gfCNCPoint2[1220] = {X 302.9698, Y 48.2613, Z -2.1667, A 0.000, B 0.000, C 0.000 }
gfCNCPoint2[1221] = {X 302.3118, Y 47.6087, Z -2.1667, A 0.000, B 0.000, C 0.000 }
gfCNCPoint2[1222] = {X 301.8147, Y 46.8265, Z -2.1667, A 0.000, B 0.000, C 0.000 }
gfCNCPoint2[1223] = {X 301.5030, Y 45.9537, Z -2.1667, A 0.000, B 0.000, C 0.000 }
gfCNCPoint2[1224] = {X 301.3924, Y 45.0335, Z -2.1667, A 0.000, B 0.000, C 0.000 }
gfCNCPoint2[1225] = {X 301.3923, Y 44.2050, Z -2.1667, A 0.000, B 0.000, C 0.000 }
gfCNCPoint2[1226] = {X 301.5103, Y 43.2839, Z -2.1667, A 0.000, B 0.000, C 0.000 }
gfCNCPoint2[1227] = {X 301.8142, Y 42.4063, Z -2.1667, A 0.000, B 0.000, C 0.000 }
gfCNCPoint2[1228] = {X 302.2910, Y 41.6094, Z -2.1667, A 0.000, B 0.000, C 0.000 }
gfCNCPoint2[1229] = {X 302.9207, Y 40.9269, Z -2.1667, A 0.000, B 0.000, C 0.000 }
gfCNCPoint2[1230] = {X 302.9207, Y 33.8743, Z -2.1667, A 0.000, B 0.000, C 0.000 }
gfCNCPoint2[1231] = {X 293.6938, Y 33.8743, Z -2.1667, A 0.000, B 0.000, C 0.000 }
gfCNCPoint2[1232] = {X 293.6927, Y 40.9767, Z -2.1667, A 0.000, B 0.000, C 0.000 }
gfCNCPoint2[1233] = {X 294.3309, Y 41.6397, Z -2.1667, A 0.000, B 0.000, C 0.000 }
gfCNCPoint2[1234] = {X 294.8119, Y 42.4241, Z -2.1667, A 0.000, B 0.000, C 0.000 }
gfCNCPoint2[1235] = {X 295.1133, Y 43.2936, Z -2.1667, A 0.000, B 0.000, C 0.000 }
gfCNCPoint2[1236] = {X 295.2211, Y 44.2074, Z -2.1667, A 0.000, B 0.000, C 0.000 }
gfCNCPoint2[1237] = {X 295.2211, Y 45.0000, Z -2.1667, A 0.000, B 0.000, C 0.000 }
gfCNCPoint2[1238] = {X 295.1168, Y 45.9257, Z -2.1667, A 0.000, B 0.000, C 0.000 }
gfCNCPoint2[1239] = {X 294.8092, Y 46.8050, Z -2.1667, A 0.000, B 0.000, C 0.000 }
gfCNCPoint2[1240] = {X 294.3136, Y 47.5937, Z -2.1667, A 0.000, B 0.000, C 0.000 }
gfCNCPoint2[1241] = {X 293.6549, Y 48.2524, Z -2.1667, A 0.000, B 0.000, C 0.000 }
gfCNCPoint2[1242] = {X 292.8661, Y 48.7480, Z -2.1667, A 0.000, B 0.000, C 0.000 }
gfCNCPoint2[1243] = {X 291.9868, Y 49.0557, Z -2.1667, A 0.000, B 0.000, C 0.000 }
gfCNCPoint2[1244] = {X 291.0611, Y 49.1600, Z -2.1667, A 0.000, B 0.000, C 0.000 }
gfCNCPoint2[1245] = {X 284.6177, Y 49.1600, Z -2.1667, A 0.000, B 0.000, C 0.000 }
gfCNCPoint2[1246] = {X 283.6967, Y 49.0568, Z -2.1667, A 0.000, B 0.000, C 0.000 }
gfCNCPoint2[1247] = {X 282.8214, Y 48.7522, Z -2.1667, A 0.000, B 0.000, C 0.000 }
gfCNCPoint2[1248] = {X 282.0353, Y 48.2615, Z -2.1667, A 0.000, B 0.000, C 0.000 }
gfCNCPoint2[1249] = {X 281.3774, Y 47.6088, Z -2.1667, A 0.000, B 0.000, C 0.000 }
gfCNCPoint2[1250] = {X 280.8802, Y 46.8267, Z -2.1667, A 0.000, B 0.000, C 0.000 }
gfCNCPoint2[1251] = {X 280.5685, Y 45.9540, Z -2.1667, A 0.000, B 0.000, C 0.000 }
gfCNCPoint2[1252] = {X 280.4578, Y 45.0339, Z -2.1667, A 0.000, B 0.000, C 0.000 }
gfCNCPoint2[1253] = {X 280.4577, Y 44.2080, Z -2.1667, A 0.000, B 0.000, C 0.000 }
gfCNCPoint2[1254] = {X 280.5632, Y 43.2953, Z -2.1667, A 0.000, B 0.000, C 0.000 }
gfCNCPoint2[1255] = {X 280.8642, Y 42.4272, Z -2.1667, A 0.000, B 0.000, C 0.000 }
gfCNCPoint2[1256] = {X 281.3461, Y 41.6449, Z -2.1667, A 0.000, B 0.000, C 0.000 }
gfCNCPoint2[1257] = {X 281.9862, Y 40.9858, Z -2.1667, A 0.000, B 0.000, C 0.000 }
gfCNCPoint2[1258] = {X 281.9860, Y 28.5930, Z -2.1667, A 0.000, B 0.000, C 0.000 }
gfCNCPoint2[1259] = {X 277.9860, Y 28.5931, Z -2.1667, A 0.000, B 0.000, C 0.000 }
gfCNCPoint2[1260] = {X 282.0660, Y 28.5930, Z -2.1667, A 0.000, B 0.000, C 0.000 }
gfCNCPoint2[1261] = {X 282.0658, Y 16.1615, Z -2.1667, A 0.000, B 0.000, C 0.000 }
gfCNCPoint2[1262] = {X 281.4285, Y 15.5227, Z -2.1667, A 0.000, B 0.000, C 0.000 }
gfCNCPoint2[1263] = {X 280.9471, Y 14.7594, Z -2.1667, A 0.000, B 0.000, C 0.000 }
gfCNCPoint2[1264] = {X 280.6453, Y 13.9090, Z -2.1667, A 0.000, B 0.000, C 0.000 }
gfCNCPoint2[1265] = {X 280.5378, Y 13.0130, Z -2.1667, A 0.000, B 0.000, C 0.000 }
gfCNCPoint2[1266] = {X 280.5377, Y 12.1868, Z -2.1667, A 0.000, B 0.000, C 0.000 }
gfCNCPoint2[1267] = {X 280.6400, Y 11.2789, Z -2.1667, A 0.000, B 0.000, C 0.000 }
gfCNCPoint2[1268] = {X 280.9417, Y 10.4166, Z -2.1667, A 0.000, B 0.000, C 0.000 }
gfCNCPoint2[1269] = {X 281.4278, Y 9.6430, Z -2.1667, A 0.000, B 0.000, C 0.000 }
gfCNCPoint2[1270] = {X 282.0738, Y 8.9969, Z -2.1667, A 0.000, B 0.000, C 0.000 }
gfCNCPoint2[1271] = {X 282.8474, Y 8.5109, Z -2.1667, A 0.000, B 0.000, C 0.000 }
gfCNCPoint2[1272] = {X 283.7098, Y 8.2091, Z -2.1667, A 0.000, B 0.000, C 0.000 }
gfCNCPoint2[1273] = {X 284.6177, Y 8.1068, Z -2.1667, A 0.000, B 0.000, C 0.000 }
gfCNCPoint2[1274] = {X 291.0611, Y 8.1068, Z -2.1667, A 0.000, B 0.000, C 0.000 }
gfCNCPoint2[1275] = {X 291.9690, Y 8.2091, Z -2.1667, A 0.000, B 0.000, C 0.000 }
gfCNCPoint2[1276] = {X 292.8314, Y 8.5109, Z -2.1667, A 0.000, B 0.000, C 0.000 }
gfCNCPoint2[1277] = {X 293.6050, Y 8.9969, Z -2.1667, A 0.000, B 0.000, C 0.000 }
gfCNCPoint2[1278] = {X 294.2510, Y 9.6430, Z -2.1667, A 0.000, B 0.000, C 0.000 }
gfCNCPoint2[1279] = {X 294.7371, Y 10.4166, Z -2.1667, A 0.000, B 0.000, C 0.000 }
gfCNCPoint2[1280] = {X 295.0388, Y 11.2789, Z -2.1667, A 0.000, B 0.000, C 0.000 }
gfCNCPoint2[1281] = {X 295.1411, Y 12.1868, Z -2.1667, A 0.000, B 0.000, C 0.000 }
gfCNCPoint2[1282] = {X 295.1411, Y 12.9781, Z -2.1667, A 0.000, B 0.000, C 0.000 }
gfCNCPoint2[1283] = {X 295.0472, Y 13.8483, Z -2.1667, A 0.000, B 0.000, C 0.000 }
gfCNCPoint2[1284] = {X 294.7699, Y 14.6784, Z -2.1667, A 0.000, B 0.000, C 0.000 }
gfCNCPoint2[1285] = {X 294.3219, Y 15.4303, Z -2.1667, A 0.000, B 0.000, C 0.000 }
gfCNCPoint2[1286] = {X 293.7238, Y 16.0694, Z -2.1667, A 0.000, B 0.000, C 0.000 }
gfCNCPoint2[1287] = {X 293.6665, Y 16.1178, Z -2.1667, A 0.000, B 0.000, C 0.000 }
gfCNCPoint2[1288] = {X 293.6084, Y 16.1652, Z -2.1667, A 0.000, B 0.000, C 0.000 }
gfCNCPoint2[1289] = {X 293.6127, Y 16.1999, Z -2.1667, A 0.000, B 0.000, C 0.000 }
gfCNCPoint2[1290] = {X 293.6140, Y 22.4371, Z -2.1667, A 0.000, B 0.000, C 0.000 }
gfCNCPoint2[1291] = {X 293.7675, Y 22.4365, Z -2.1667, A 0.000, B 0.000, C 0.000 }
gfCNCPoint2[1292] = {X 302.9997, Y 22.4365, Z -2.1667, A 0.000, B 0.000, C 0.000 }
gfCNCPoint2[1293] = {X 303.0047, Y 16.1649, Z -2.1667, A 0.000, B 0.000, C 0.000 }
gfCNCPoint2[1294] = {X 302.9465, Y 16.1175, Z -2.1667, A 0.000, B 0.000, C 0.000 }
gfCNCPoint2[1295] = {X 302.8892, Y 16.0690, Z -2.1667, A 0.000, B 0.000, C 0.000 }
gfCNCPoint2[1296] = {X 302.2967, Y 15.4373, Z -2.1667, A 0.000, B 0.000, C 0.000 }
gfCNCPoint2[1297] = {X 301.8510, Y 14.6947, Z -2.1667, A 0.000, B 0.000, C 0.000 }
gfCNCPoint2[1298] = {X 301.5720, Y 13.8747, Z -2.1667, A 0.000, B 0.000, C 0.000 }
gfCNCPoint2[1299] = {X 301.4724, Y 13.0144, Z -2.1667, A 0.000, B 0.000, C 0.000 }
gfCNCPoint2[1300] = {X 301.4723, Y 12.1868, Z -2.1667, A 0.000, B 0.000, C 0.000 }
gfCNCPoint2[1301] = {X 301.5745, Y 11.2789, Z -2.1667, A 0.000, B 0.000, C 0.000 }
gfCNCPoint2[1302] = {X 301.8763, Y 10.4166, Z -2.1667, A 0.000, B 0.000, C 0.000 }
gfCNCPoint2[1303] = {X 302.3624, Y 9.6430, Z -2.1667, A 0.000, B 0.000, C 0.000 }
gfCNCPoint2[1304] = {X 303.0084, Y 8.9969, Z -2.1667, A 0.000, B 0.000, C 0.000 }
gfCNCPoint2[1305] = {X 303.7820, Y 8.5109, Z -2.1667, A 0.000, B 0.000, C 0.000 }
gfCNCPoint2[1306] = {X 304.6444, Y 8.2091, Z -2.1667, A 0.000, B 0.000, C 0.000 }
gfCNCPoint2[1307] = {X 305.5523, Y 8.1068, Z -2.1667, A 0.000, B 0.000, C 0.000 }
gfCNCPoint2[1308] = {X 311.9957, Y 8.1068, Z -2.1667, A 0.000, B 0.000, C 0.000 }
gfCNCPoint2[1309] = {X 312.9036, Y 8.2091, Z -2.1667, A 0.000, B 0.000, C 0.000 }
gfCNCPoint2[1310] = {X 313.7660, Y 8.5109, Z -2.1667, A 0.000, B 0.000, C 0.000 }
gfCNCPoint2[1311] = {X 314.5396, Y 8.9969, Z -2.1667, A 0.000, B 0.000, C 0.000 }
gfCNCPoint2[1312] = {X 315.1856, Y 9.6430, Z -2.1667, A 0.000, B 0.000, C 0.000 }
gfCNCPoint2[1313] = {X 315.6717, Y 10.4166, Z -2.1667, A 0.000, B 0.000, C 0.000 }
gfCNCPoint2[1314] = {X 315.9734, Y 11.2789, Z -2.1667, A 0.000, B 0.000, C 0.000 }
gfCNCPoint2[1315] = {X 316.0757, Y 12.1868, Z -2.1667, A 0.000, B 0.000, C 0.000 }
gfCNCPoint2[1316] = {X 316.0757, Y 12.9781, Z -2.1667, A 0.000, B 0.000, C 0.000 }
gfCNCPoint2[1317] = {X 315.9818, Y 13.8483, Z -2.1667, A 0.000, B 0.000, C 0.000 }
gfCNCPoint2[1318] = {X 315.7045, Y 14.6784, Z -2.1667, A 0.000, B 0.000, C 0.000 }
gfCNCPoint2[1319] = {X 315.2566, Y 15.4302, Z -2.1667, A 0.000, B 0.000, C 0.000 }
gfCNCPoint2[1320] = {X 314.6586, Y 16.0692, Z -2.1667, A 0.000, B 0.000, C 0.000 }
gfCNCPoint2[1321] = {X 314.6041, Y 16.1153, Z -2.1667, A 0.000, B 0.000, C 0.000 }
gfCNCPoint2[1322] = {X 314.5488, Y 16.1605, Z -2.1667, A 0.000, B 0.000, C 0.000 }
gfCNCPoint2[1323] = {X 314.5472, Y 41.0281, Z -2.1667, A 0.000, B 0.000, C 0.000 }
gfCNCPoint2[1324] = {X 314.6336, Y 41.0962, Z -2.1667, A 0.000, B 0.000, C 0.000 }
gfCNCPoint2[1325] = {X 315.2363, Y 41.7299, Z -2.1667, A 0.000, B 0.000, C 0.000 }
gfCNCPoint2[1326] = {X 315.6902, Y 42.4775, Z -2.1667, A 0.000, B 0.000, C 0.000 }
gfCNCPoint2[1327] = {X 315.9743, Y 43.3047, Z -2.1667, A 0.000, B 0.000, C 0.000 }
gfCNCPoint2[1328] = {X 316.0756, Y 44.1734, Z -2.1667, A 0.000, B 0.000, C 0.000 }
gfCNCPoint2[1329] = {X 316.0757, Y 45.0000, Z -2.1667, A 0.000, B 0.000, C 0.000 }
gfCNCPoint2[1330] = {X 315.9734, Y 45.9079, Z -2.1667, A 0.000, B 0.000, C 0.000 }
gfCNCPoint2[1331] = {X 315.6717, Y 46.7702, Z -2.1667, A 0.000, B 0.000, C 0.000 }
gfCNCPoint2[1332] = {X 315.1856, Y 47.5438, Z -2.1667, A 0.000, B 0.000, C 0.000 }
gfCNCPoint2[1333] = {X 314.5396, Y 48.1899, Z -2.1667, A 0.000, B 0.000, C 0.000 }
gfCNCPoint2[1334] = {X 313.7660, Y 48.6760, Z -2.1667, A 0.000, B 0.000, C 0.000 }
gfCNCPoint2[1335] = {X 312.9036, Y 48.9777, Z -2.1667, A 0.000, B 0.000, C 0.000 }
gfCNCPoint2[1336] = {X 311.9957, Y 49.0800, Z -2.1667, A 0.000, B 0.000, C 0.000 }
gfCNCPoint2[1337] = {X 305.5523, Y 49.0800, Z -2.1667, A 0.000, B 0.000, C 0.000 }
gfCNCPoint2[1338] = {X 304.6489, Y 48.9787, Z -2.1667, A 0.000, B 0.000, C 0.000 }
gfCNCPoint2[1339] = {X 303.7905, Y 48.6800, Z -2.1667, A 0.000, B 0.000, C 0.000 }
gfCNCPoint2[1340] = {X 303.0194, Y 48.1986, Z -2.1667, A 0.000, B 0.000, C 0.000 }
gfCNCPoint2[1341] = {X 302.3741, Y 47.5585, Z -2.1667, A 0.000, B 0.000, C 0.000 }
gfCNCPoint2[1342] = {X 301.8865, Y 46.7914, Z -2.1667, A 0.000, B 0.000, C 0.000 }
gfCNCPoint2[1343] = {X 301.5809, Y 45.9353, Z -2.1667, A 0.000, B 0.000, C 0.000 }
gfCNCPoint2[1344] = {X 301.4724, Y 45.0328, Z -2.1667, A 0.000, B 0.000, C 0.000 }
gfCNCPoint2[1345] = {X 301.4723, Y 44.2070, Z -2.1667, A 0.000, B 0.000, C 0.000 }
gfCNCPoint2[1346] = {X 301.5903, Y 43.2934, Z -2.1667, A 0.000, B 0.000, C 0.000 }
gfCNCPoint2[1347] = {X 301.8943, Y 42.4238, Z -2.1667, A 0.000, B 0.000, C 0.000 }
gfCNCPoint2[1348] = {X 302.3713, Y 41.6358, Z -2.1667, A 0.000, B 0.000, C 0.000 }
gfCNCPoint2[1349] = {X 303.0007, Y 40.9632, Z -2.1667, A 0.000, B 0.000, C 0.000 }
gfCNCPoint2[1350] = {X 303.0007, Y 33.7943, Z -2.1667, A 0.000, B 0.000, C 0.000 }
gfCNCPoint2[1351] = {X 293.6138, Y 33.7943, Z -2.1667, A 0.000, B 0.000, C 0.000 }
gfCNCPoint2[1352] = {X 293.6127, Y 41.0143, Z -2.1667, A 0.000, B 0.000, C 0.000 }
gfCNCPoint2[1353] = {X 294.2505, Y 41.6665, Z -2.1667, A 0.000, B 0.000, C 0.000 }
gfCNCPoint2[1354] = {X 294.7316, Y 42.4415, Z -2.1667, A 0.000, B 0.000, C 0.000 }
gfCNCPoint2[1355] = {X 295.0333, Y 43.3024, Z -2.1667, A 0.000, B 0.000, C 0.000 }
gfCNCPoint2[1356] = {X 295.1411, Y 44.2082, Z -2.1667, A 0.000, B 0.000, C 0.000 }
gfCNCPoint2[1357] = {X 295.1411, Y 45.0000, Z -2.1667, A 0.000, B 0.000, C 0.000 }
gfCNCPoint2[1358] = {X 295.0388, Y 45.9079, Z -2.1667, A 0.000, B 0.000, C 0.000 }
gfCNCPoint2[1359] = {X 294.7371, Y 46.7702, Z -2.1667, A 0.000, B 0.000, C 0.000 }
gfCNCPoint2[1360] = {X 294.2510, Y 47.5438, Z -2.1667, A 0.000, B 0.000, C 0.000 }
gfCNCPoint2[1361] = {X 293.6050, Y 48.1899, Z -2.1667, A 0.000, B 0.000, C 0.000 }
gfCNCPoint2[1362] = {X 292.8314, Y 48.6760, Z -2.1667, A 0.000, B 0.000, C 0.000 }
gfCNCPoint2[1363] = {X 291.9690, Y 48.9777, Z -2.1667, A 0.000, B 0.000, C 0.000 }
gfCNCPoint2[1364] = {X 291.0611, Y 49.0800, Z -2.1667, A 0.000, B 0.000, C 0.000 }
gfCNCPoint2[1365] = {X 284.6177, Y 49.0800, Z -2.1667, A 0.000, B 0.000, C 0.000 }
gfCNCPoint2[1366] = {X 283.7144, Y 48.9788, Z -2.1667, A 0.000, B 0.000, C 0.000 }
gfCNCPoint2[1367] = {X 282.8560, Y 48.6801, Z -2.1667, A 0.000, B 0.000, C 0.000 }
gfCNCPoint2[1368] = {X 282.0850, Y 48.1987, Z -2.1667, A 0.000, B 0.000, C 0.000 }
gfCNCPoint2[1369] = {X 281.4397, Y 47.5587, Z -2.1667, A 0.000, B 0.000, C 0.000 }
gfCNCPoint2[1370] = {X 280.9521, Y 46.7916, Z -2.1667, A 0.000, B 0.000, C 0.000 }
gfCNCPoint2[1371] = {X 280.6464, Y 45.9356, Z -2.1667, A 0.000, B 0.000, C 0.000 }
gfCNCPoint2[1372] = {X 280.5378, Y 45.0332, Z -2.1667, A 0.000, B 0.000, C 0.000 }
gfCNCPoint2[1373] = {X 280.5377, Y 44.2084, Z -2.1667, A 0.000, B 0.000, C 0.000 }
gfCNCPoint2[1374] = {X 280.6433, Y 43.3039, Z -2.1667, A 0.000, B 0.000, C 0.000 }
gfCNCPoint2[1375] = {X 280.9445, Y 42.4445, Z -2.1667, A 0.000, B 0.000, C 0.000 }
gfCNCPoint2[1376] = {X 281.4266, Y 41.6719, Z -2.1667, A 0.000, B 0.000, C 0.000 }
gfCNCPoint2[1377] = {X 282.0662, Y 41.0237, Z -2.1667, A 0.000, B 0.000, C 0.000 }
gfCNCPoint2[1378] = {X 282.0660, Y 28.5930, Z -2.1667, A 0.000, B 0.000, C 0.000 }
gfCNCPoint2[1379] = {X 278.0660, Y 28.5931, Z -2.1667, A 0.000, B 0.000, C 0.000 }
gfCNCPoint2[1380] = {X 282.1460, Y 28.5930, Z -2.1667, A 0.000, B 0.000, C 0.000 }
gfCNCPoint2[1381] = {X 282.1458, Y 16.1228, Z -2.1667, A 0.000, B 0.000, C 0.000 }
gfCNCPoint2[1382] = {X 281.5036, Y 15.4885, Z -2.1667, A 0.000, B 0.000, C 0.000 }
gfCNCPoint2[1383] = {X 281.0199, Y 14.7262, Z -2.1667, A 0.000, B 0.000, C 0.000 }
gfCNCPoint2[1384] = {X 280.7195, Y 13.8749, Z -2.1667, A 0.000, B 0.000, C 0.000 }
gfCNCPoint2[1385] = {X 280.6177, Y 12.9779, Z -2.1667, A 0.000, B 0.000, C 0.000 }
gfCNCPoint2[1386] = {X 280.6177, Y 12.1868, Z -2.1667, A 0.000, B 0.000, C 0.000 }
gfCNCPoint2[1387] = {X 280.7180, Y 11.2967, Z -2.1667, A 0.000, B 0.000, C 0.000 }
gfCNCPoint2[1388] = {X 281.0138, Y 10.4513, Z -2.1667, A 0.000, B 0.000, C 0.000 }
gfCNCPoint2[1389] = {X 281.4903, Y 9.6929, Z -2.1667, A 0.000, B 0.000, C 0.000 }
gfCNCPoint2[1390] = {X 282.1237, Y 9.0595, Z -2.1667, A 0.000, B 0.000, C 0.000 }
gfCNCPoint2[1391] = {X 282.8821, Y 8.5829, Z -2.1667, A 0.000, B 0.000, C 0.000 }
gfCNCPoint2[1392] = {X 283.7276, Y 8.2871, Z -2.1667, A 0.000, B 0.000, C 0.000 }
gfCNCPoint2[1393] = {X 284.6177, Y 8.1868, Z -2.1667, A 0.000, B 0.000, C 0.000 }
gfCNCPoint2[1394] = {X 291.0611, Y 8.1868, Z -2.1667, A 0.000, B 0.000, C 0.000 }
gfCNCPoint2[1395] = {X 291.9512, Y 8.2871, Z -2.1667, A 0.000, B 0.000, C 0.000 }
gfCNCPoint2[1396] = {X 292.7967, Y 8.5829, Z -2.1667, A 0.000, B 0.000, C 0.000 }
gfCNCPoint2[1397] = {X 293.5551, Y 9.0595, Z -2.1667, A 0.000, B 0.000, C 0.000 }
gfCNCPoint2[1398] = {X 294.1885, Y 9.6929, Z -2.1667, A 0.000, B 0.000, C 0.000 }
gfCNCPoint2[1399] = {X 294.6650, Y 10.4513, Z -2.1667, A 0.000, B 0.000, C 0.000 }
gfCNCPoint2[1400] = {X 294.9608, Y 11.2967, Z -2.1667, A 0.000, B 0.000, C 0.000 }
gfCNCPoint2[1401] = {X 295.0611, Y 12.1868, Z -2.1667, A 0.000, B 0.000, C 0.000 }
gfCNCPoint2[1402] = {X 295.0609, Y 13.0192, Z -2.1667, A 0.000, B 0.000, C 0.000 }
gfCNCPoint2[1403] = {X 294.9624, Y 13.8613, Z -2.1667, A 0.000, B 0.000, C 0.000 }
gfCNCPoint2[1404] = {X 294.6886, Y 14.6637, Z -2.1667, A 0.000, B 0.000, C 0.000 }
gfCNCPoint2[1405] = {X 294.2518, Y 15.3904, Z -2.1667, A 0.000, B 0.000, C 0.000 }
gfCNCPoint2[1406] = {X 293.6716, Y 16.0087, Z -2.1667, A 0.000, B 0.000, C 0.000 }
gfCNCPoint2[1407] = {X 293.5954, Y 16.0727, Z -2.1667, A 0.000, B 0.000, C 0.000 }
gfCNCPoint2[1408] = {X 293.5177, Y 16.1348, Z -2.1667, A 0.000, B 0.000, C 0.000 }
gfCNCPoint2[1409] = {X 293.5327, Y 16.1919, Z -2.1667, A 0.000, B 0.000, C 0.000 }
gfCNCPoint2[1410] = {X 293.5341, Y 22.5174, Z -2.1667, A 0.000, B 0.000, C 0.000 }
gfCNCPoint2[1411] = {X 293.7676, Y 22.5165, Z -2.1667, A 0.000, B 0.000, C 0.000 }
gfCNCPoint2[1412] = {X 303.0796, Y 22.5177, Z -2.1667, A 0.000, B 0.000, C 0.000 }
gfCNCPoint2[1413] = {X 303.0803, Y 16.1920, Z -2.1667, A 0.000, B 0.000, C 0.000 }
gfCNCPoint2[1414] = {X 303.0955, Y 16.1346, Z -2.1667, A 0.000, B 0.000, C 0.000 }
gfCNCPoint2[1415] = {X 303.0176, Y 16.0725, Z -2.1667, A 0.000, B 0.000, C 0.000 }
gfCNCPoint2[1416] = {X 302.9414, Y 16.0084, Z -2.1667, A 0.000, B 0.000, C 0.000 }
gfCNCPoint2[1417] = {X 302.3552, Y 15.3819, Z -2.1667, A 0.000, B 0.000, C 0.000 }
gfCNCPoint2[1418] = {X 301.9161, Y 14.6448, Z -2.1667, A 0.000, B 0.000, C 0.000 }
gfCNCPoint2[1419] = {X 301.6443, Y 13.8310, Z -2.1667, A 0.000, B 0.000, C 0.000 }
gfCNCPoint2[1420] = {X 301.5523, Y 12.9779, Z -2.1667, A 0.000, B 0.000, C 0.000 }
gfCNCPoint2[1421] = {X 301.5523, Y 12.1868, Z -2.1667, A 0.000, B 0.000, C 0.000 }
gfCNCPoint2[1422] = {X 301.6525, Y 11.2967, Z -2.1667, A 0.000, B 0.000, C 0.000 }
gfCNCPoint2[1423] = {X 301.9484, Y 10.4513, Z -2.1667, A 0.000, B 0.000, C 0.000 }
gfCNCPoint2[1424] = {X 302.4249, Y 9.6929, Z -2.1667, A 0.000, B 0.000, C 0.000 }
gfCNCPoint2[1425] = {X 303.0583, Y 9.0595, Z -2.1667, A 0.000, B 0.000, C 0.000 }
gfCNCPoint2[1426] = {X 303.8167, Y 8.5829, Z -2.1667, A 0.000, B 0.000, C 0.000 }
gfCNCPoint2[1427] = {X 304.6622, Y 8.2871, Z -2.1667, A 0.000, B 0.000, C 0.000 }
gfCNCPoint2[1428] = {X 305.5523, Y 8.1868, Z -2.1667, A 0.000, B 0.000, C 0.000 }
gfCNCPoint2[1429] = {X 311.9957, Y 8.1868, Z -2.1667, A 0.000, B 0.000, C 0.000 }
gfCNCPoint2[1430] = {X 312.8858, Y 8.2871, Z -2.1667, A 0.000, B 0.000, C 0.000 }
gfCNCPoint2[1431] = {X 313.7313, Y 8.5829, Z -2.1667, A 0.000, B 0.000, C 0.000 }
gfCNCPoint2[1432] = {X 314.4897, Y 9.0595, Z -2.1667, A 0.000, B 0.000, C 0.000 }
gfCNCPoint2[1433] = {X 315.1230, Y 9.6929, Z -2.1667, A 0.000, B 0.000, C 0.000 }
gfCNCPoint2[1434] = {X 315.5996, Y 10.4513, Z -2.1667, A 0.000, B 0.000, C 0.000 }
gfCNCPoint2[1435] = {X 315.8954, Y 11.2967, Z -2.1667, A 0.000, B 0.000, C 0.000 }
gfCNCPoint2[1436] = {X 315.9957, Y 12.1868, Z -2.1667, A 0.000, B 0.000, C 0.000 }
gfCNCPoint2[1437] = {X 315.9955, Y 13.0192, Z -2.1667, A 0.000, B 0.000, C 0.000 }
gfCNCPoint2[1438] = {X 315.8970, Y 13.8613, Z -2.1667, A 0.000, B 0.000, C 0.000 }
gfCNCPoint2[1439] = {X 315.6232, Y 14.6637, Z -2.1667, A 0.000, B 0.000, C 0.000 }
gfCNCPoint2[1440] = {X 315.1865, Y 15.3903, Z -2.1667, A 0.000, B 0.000, C 0.000 }
gfCNCPoint2[1441] = {X 314.6064, Y 16.0086, Z -2.1667, A 0.000, B 0.000, C 0.000 }
gfCNCPoint2[1442] = {X 314.5386, Y 16.0657, Z -2.1667, A 0.000, B 0.000, C 0.000 }
gfCNCPoint2[1443] = {X 314.4695, Y 16.1213, Z -2.1667, A 0.000, B 0.000, C 0.000 }
gfCNCPoint2[1444] = {X 314.4674, Y 16.3117, Z -2.1667, A 0.000, B 0.000, C 0.000 }
gfCNCPoint2[1445] = {X 314.4672, Y 41.0669, Z -2.1667, A 0.000, B 0.000, C 0.000 }
gfCNCPoint2[1446] = {X 314.6061, Y 41.1780, Z -2.1667, A 0.000, B 0.000, C 0.000 }
gfCNCPoint2[1447] = {X 315.1925, Y 41.8046, Z -2.1667, A 0.000, B 0.000, C 0.000 }
gfCNCPoint2[1448] = {X 315.6318, Y 42.5418, Z -2.1667, A 0.000, B 0.000, C 0.000 }
gfCNCPoint2[1449] = {X 315.9037, Y 43.3557, Z -2.1667, A 0.000, B 0.000, C 0.000 }
gfCNCPoint2[1450] = {X 315.9957, Y 44.2089, Z -2.1667, A 0.000, B 0.000, C 0.000 }
gfCNCPoint2[1451] = {X 315.9957, Y 45.0000, Z -2.1667, A 0.000, B 0.000, C 0.000 }
gfCNCPoint2[1452] = {X 315.8954, Y 45.8901, Z -2.1667, A 0.000, B 0.000, C 0.000 }
gfCNCPoint2[1453] = {X 315.5996, Y 46.7355, Z -2.1667, A 0.000, B 0.000, C 0.000 }
gfCNCPoint2[1454] = {X 315.1230, Y 47.4940, Z -2.1667, A 0.000, B 0.000, C 0.000 }
gfCNCPoint2[1455] = {X 314.4897, Y 48.1273, Z -2.1667, A 0.000, B 0.000, C 0.000 }
gfCNCPoint2[1456] = {X 313.7313, Y 48.6039, Z -2.1667, A 0.000, B 0.000, C 0.000 }
gfCNCPoint2[1457] = {X 312.8858, Y 48.8997, Z -2.1667, A 0.000, B 0.000, C 0.000 }
gfCNCPoint2[1458] = {X 311.9957, Y 49.0000, Z -2.1667, A 0.000, B 0.000, C 0.000 }
gfCNCPoint2[1459] = {X 305.5523, Y 49.0000, Z -2.1667, A 0.000, B 0.000, C 0.000 }
gfCNCPoint2[1460] = {X 304.6622, Y 48.8997, Z -2.1667, A 0.000, B 0.000, C 0.000 }
gfCNCPoint2[1461] = {X 303.8167, Y 48.6039, Z -2.1667, A 0.000, B 0.000, C 0.000 }
gfCNCPoint2[1462] = {X 303.0583, Y 48.1273, Z -2.1667, A 0.000, B 0.000, C 0.000 }
gfCNCPoint2[1463] = {X 302.4249, Y 47.4939, Z -2.1667, A 0.000, B 0.000, C 0.000 }
gfCNCPoint2[1464] = {X 301.9484, Y 46.7355, Z -2.1667, A 0.000, B 0.000, C 0.000 }
gfCNCPoint2[1465] = {X 301.6525, Y 45.8900, Z -2.1667, A 0.000, B 0.000, C 0.000 }
gfCNCPoint2[1466] = {X 301.5523, Y 45.0000, Z -2.1667, A 0.000, B 0.000, C 0.000 }
gfCNCPoint2[1467] = {X 301.5523, Y 44.2089, Z -2.1667, A 0.000, B 0.000, C 0.000 }
gfCNCPoint2[1468] = {X 301.6702, Y 43.3029, Z -2.1667, A 0.000, B 0.000, C 0.000 }
gfCNCPoint2[1469] = {X 301.9745, Y 42.4415, Z -2.1667, A 0.000, B 0.000, C 0.000 }
gfCNCPoint2[1470] = {X 302.4516, Y 41.6624, Z -2.1667, A 0.000, B 0.000, C 0.000 }
gfCNCPoint2[1471] = {X 303.0807, Y 40.9999, Z -2.1667, A 0.000, B 0.000, C 0.000 }
gfCNCPoint2[1472] = {X 303.0807, Y 33.7143, Z -2.1667, A 0.000, B 0.000, C 0.000 }
gfCNCPoint2[1473] = {X 293.9337, Y 33.7143, Z -2.1667, A 0.000, B 0.000, C 0.000 }
gfCNCPoint2[1474] = {X 293.5338, Y 33.7132, Z -2.1667, A 0.000, B 0.000, C 0.000 }
gfCNCPoint2[1475] = {X 293.5327, Y 41.0524, Z -2.1667, A 0.000, B 0.000, C 0.000 }
gfCNCPoint2[1476] = {X 294.1700, Y 41.6937, Z -2.1667, A 0.000, B 0.000, C 0.000 }
gfCNCPoint2[1477] = {X 294.6513, Y 42.4591, Z -2.1667, A 0.000, B 0.000, C 0.000 }
gfCNCPoint2[1478] = {X 294.9532, Y 43.3113, Z -2.1667, A 0.000, B 0.000, C 0.000 }
gfCNCPoint2[1479] = {X 295.0611, Y 44.2089, Z -2.1667, A 0.000, B 0.000, C 0.000 }
gfCNCPoint2[1480] = {X 295.0611, Y 45.0000, Z -2.1667, A 0.000, B 0.000, C 0.000 }
gfCNCPoint2[1481] = {X 294.9608, Y 45.8901, Z -2.1667, A 0.000, B 0.000, C 0.000 }
gfCNCPoint2[1482] = {X 294.6650, Y 46.7355, Z -2.1667, A 0.000, B 0.000, C 0.000 }
gfCNCPoint2[1483] = {X 294.1885, Y 47.4940, Z -2.1667, A 0.000, B 0.000, C 0.000 }
gfCNCPoint2[1484] = {X 293.5551, Y 48.1273, Z -2.1667, A 0.000, B 0.000, C 0.000 }
gfCNCPoint2[1485] = {X 292.7967, Y 48.6039, Z -2.1667, A 0.000, B 0.000, C 0.000 }
gfCNCPoint2[1486] = {X 291.9512, Y 48.8997, Z -2.1667, A 0.000, B 0.000, C 0.000 }
gfCNCPoint2[1487] = {X 291.0611, Y 49.0000, Z -2.1667, A 0.000, B 0.000, C 0.000 }
gfCNCPoint2[1488] = {X 284.6177, Y 49.0000, Z -2.1667, A 0.000, B 0.000, C 0.000 }
gfCNCPoint2[1489] = {X 283.7276, Y 48.8997, Z -2.1667, A 0.000, B 0.000, C 0.000 }
gfCNCPoint2[1490] = {X 282.8821, Y 48.6039, Z -2.1667, A 0.000, B 0.000, C 0.000 }
gfCNCPoint2[1491] = {X 282.1237, Y 48.1273, Z -2.1667, A 0.000, B 0.000, C 0.000 }
gfCNCPoint2[1492] = {X 281.4903, Y 47.4939, Z -2.1667, A 0.000, B 0.000, C 0.000 }
gfCNCPoint2[1493] = {X 281.0138, Y 46.7355, Z -2.1667, A 0.000, B 0.000, C 0.000 }
gfCNCPoint2[1494] = {X 280.7179, Y 45.8900, Z -2.1667, A 0.000, B 0.000, C 0.000 }
gfCNCPoint2[1495] = {X 280.6177, Y 45.0000, Z -2.1667, A 0.000, B 0.000, C 0.000 }
gfCNCPoint2[1496] = {X 280.6177, Y 44.2089, Z -2.1667, A 0.000, B 0.000, C 0.000 }
gfCNCPoint2[1497] = {X 280.7234, Y 43.3127, Z -2.1667, A 0.000, B 0.000, C 0.000 }
gfCNCPoint2[1498] = {X 281.0249, Y 42.4620, Z -2.1667, A 0.000, B 0.000, C 0.000 }
gfCNCPoint2[1499] = {X 281.5071, Y 41.6992, Z -2.1667, A 0.000, B 0.000, C 0.000 }
gfCNCPoint2[1500] = {X 282.1462, Y 41.0620, Z -2.1667, A 0.000, B 0.000, C 0.000 }
gfCNCPoint2[1501] = {X 282.1460, Y 28.5930, Z -2.1667, A 0.000, B 0.000, C 0.000 }
gfCNCPoint2[1502] = {X 278.0660, Y 28.5931, Z -2.1667, A 0.000, B 0.000, C 0.000 }
gfCNCPoint2[1503] = {X 278.0660, Y 28.5931, Z 0.8333, A 0.000, B 0.000, C 0.000 }
gfCNCPoint2[1504] = {X 278.0660, Y 28.5931, Z 11.0000, A 0.000, B 0.000, C 0.000 }
gfCNCPoint2[1505] = {X 353.3541, Y 107.0427, Z 11.0000, A 0.000, B 0.000, C 0.000 }
gfCNCPoint2[1506] = {X 353.3541, Y 107.0427, Z 0.8333, A 0.000, B 0.000, C 0.000 }
gfCNCPoint2[1507] = {X 353.3541, Y 107.0427, Z -2.1667, A 0.000, B 0.000, C 0.000 }
gfCNCPoint2[1508] = {X 353.2424, Y 102.9642, Z -2.1667, A 0.000, B 0.000, C 0.000 }
gfCNCPoint2[1509] = {X 347.7202, Y 103.0327, Z -2.1667, A 0.000, B 0.000, C 0.000 }
gfCNCPoint2[1510] = {X 342.1984, Y 102.9360, Z -2.1667, A 0.000, B 0.000, C 0.000 }
gfCNCPoint2[1511] = {X 336.6820, Y 102.6741, Z -2.1667, A 0.000, B 0.000, C 0.000 }
gfCNCPoint2[1512] = {X 333.1921, Y 102.3991, Z -2.1667, A 0.000, B 0.000, C 0.000 }
gfCNCPoint2[1513] = {X 329.7159, Y 101.9862, Z -2.1667, A 0.000, B 0.000, C 0.000 }
gfCNCPoint2[1514] = {X 326.2587, Y 101.4359, Z -2.1667, A 0.000, B 0.000, C 0.000 }
gfCNCPoint2[1515] = {X 323.4092, Y 100.8312, Z -2.1667, A 0.000, B 0.000, C 0.000 }
gfCNCPoint2[1516] = {X 320.6119, Y 100.0183, Z -2.1667, A 0.000, B 0.000, C 0.000 }
gfCNCPoint2[1517] = {X 317.8822, Y 99.0016, Z -2.1667, A 0.000, B 0.000, C 0.000 }
gfCNCPoint2[1518] = {X 316.3696, Y 98.3034, Z -2.1667, A 0.000, B 0.000, C 0.000 }
gfCNCPoint2[1519] = {X 314.9205, Y 97.4815, Z -2.1667, A 0.000, B 0.000, C 0.000 }
gfCNCPoint2[1520] = {X 313.5450, Y 96.5415, Z -2.1667, A 0.000, B 0.000, C 0.000 }
gfCNCPoint2[1521] = {X 312.2527, Y 95.4901, Z -2.1667, A 0.000, B 0.000, C 0.000 }
gfCNCPoint2[1522] = {X 311.2490, Y 94.4920, Z -2.1667, A 0.000, B 0.000, C 0.000 }
gfCNCPoint2[1523] = {X 310.3708, Y 93.3817, Z -2.1667, A 0.000, B 0.000, C 0.000 }
gfCNCPoint2[1524] = {X 309.6305, Y 92.1752, Z -2.1667, A 0.000, B 0.000, C 0.000 }
gfCNCPoint2[1525] = {X 309.0387, Y 90.8892, Z -2.1667, A 0.000, B 0.000, C 0.000 }
gfCNCPoint2[1526] = {X 308.6036, Y 89.5422, Z -2.1667, A 0.000, B 0.000, C 0.000 }
gfCNCPoint2[1527] = {X 308.2601, Y 87.9191, Z -2.1667, A 0.000, B 0.000, C 0.000 }
gfCNCPoint2[1528] = {X 308.0572, Y 86.2724, Z -2.1667, A 0.000, B 0.000, C 0.000 }
gfCNCPoint2[1529] = {X 307.9964, Y 84.6145, Z -2.1667, A 0.000, B 0.000, C 0.000 }
gfCNCPoint2[1530] = {X 307.9976, Y 83.2310, Z -2.1667, A 0.000, B 0.000, C 0.000 }
gfCNCPoint2[1531] = {X 307.9976, Y 63.2124, Z -2.1667, A 0.000, B 0.000, C 0.000 }
gfCNCPoint2[1532] = {X 307.1459, Y 63.0033, Z -2.1667, A 0.000, B 0.000, C 0.000 }
gfCNCPoint2[1533] = {X 306.3540, Y 62.6266, Z -2.1667, A 0.000, B 0.000, C 0.000 }
gfCNCPoint2[1534] = {X 305.6544, Y 62.0976, Z -2.1667, A 0.000, B 0.000, C 0.000 }
gfCNCPoint2[1535] = {X 305.0761, Y 61.4383, Z -2.1667, A 0.000, B 0.000, C 0.000 }
gfCNCPoint2[1536] = {X 304.6429, Y 60.6758, Z -2.1667, A 0.000, B 0.000, C 0.000 }
gfCNCPoint2[1537] = {X 304.3726, Y 59.8415, Z -2.1667, A 0.000, B 0.000, C 0.000 }
gfCNCPoint2[1538] = {X 304.2764, Y 58.9697, Z -2.1667, A 0.000, B 0.000, C 0.000 }
gfCNCPoint2[1539] = {X 304.2762, Y 58.0000, Z -2.1667, A 0.000, B 0.000, C 0.000 }
gfCNCPoint2[1540] = {X 304.3845, Y 57.0387, Z -2.1667, A 0.000, B 0.000, C 0.000 }
gfCNCPoint2[1541] = {X 304.7040, Y 56.1256, Z -2.1667, A 0.000, B 0.000, C 0.000 }
gfCNCPoint2[1542] = {X 305.2187, Y 55.3065, Z -2.1667, A 0.000, B 0.000, C 0.000 }
gfCNCPoint2[1543] = {X 305.9027, Y 54.6225, Z -2.1667, A 0.000, B 0.000, C 0.000 }
gfCNCPoint2[1544] = {X 306.7218, Y 54.1078, Z -2.1667, A 0.000, B 0.000, C 0.000 }
gfCNCPoint2[1545] = {X 307.6349, Y 53.7883, Z -2.1667, A 0.000, B 0.000, C 0.000 }
gfCNCPoint2[1546] = {X 308.5962, Y 53.6800, Z -2.1667, A 0.000, B 0.000, C 0.000 }
gfCNCPoint2[1547] = {X 324.3107, Y 53.6800, Z -2.1667, A 0.000, B 0.000, C 0.000 }
gfCNCPoint2[1548] = {X 325.2720, Y 53.7883, Z -2.1667, A 0.000, B 0.000, C 0.000 }
gfCNCPoint2[1549] = {X 326.1851, Y 54.1078, Z -2.1667, A 0.000, B 0.000, C 0.000 }
gfCNCPoint2[1550] = {X 327.0042, Y 54.6225, Z -2.1667, A 0.000, B 0.000, C 0.000 }
gfCNCPoint2[1551] = {X 327.6882, Y 55.3065, Z -2.1667, A 0.000, B 0.000, C 0.000 }
gfCNCPoint2[1552] = {X 328.2029, Y 56.1256, Z -2.1667, A 0.000, B 0.000, C 0.000 }
gfCNCPoint2[1553] = {X 328.5224, Y 57.0387, Z -2.1667, A 0.000, B 0.000, C 0.000 }
gfCNCPoint2[1554] = {X 328.6307, Y 58.0000, Z -2.1667, A 0.000, B 0.000, C 0.000 }
gfCNCPoint2[1555] = {X 328.6307, Y 58.9361, Z -2.1667, A 0.000, B 0.000, C 0.000 }
gfCNCPoint2[1556] = {X 328.5362, Y 59.8122, Z -2.1667, A 0.000, B 0.000, C 0.000 }
gfCNCPoint2[1557] = {X 328.2675, Y 60.6515, Z -2.1667, A 0.000, B 0.000, C 0.000 }
gfCNCPoint2[1558] = {X 327.8355, Y 61.4196, Z -2.1667, A 0.000, B 0.000, C 0.000 }
gfCNCPoint2[1559] = {X 327.2578, Y 62.0851, Z -2.1667, A 0.000, B 0.000, C 0.000 }
gfCNCPoint2[1560] = {X 326.5581, Y 62.6208, Z -2.1667, A 0.000, B 0.000, C 0.000 }
gfCNCPoint2[1561] = {X 325.7650, Y 63.0049, Z -2.1667, A 0.000, B 0.000, C 0.000 }
gfCNCPoint2[1562] = {X 324.9108, Y 63.2217, Z -2.1667, A 0.000, B 0.000, C 0.000 }
gfCNCPoint2[1563] = {X 324.9122, Y 83.2296, Z -2.1667, A 0.000, B 0.000, C 0.000 }
gfCNCPoint2[1564] = {X 324.9258, Y 84.6149, Z -2.1667, A 0.000, B 0.000, C 0.000 }
gfCNCPoint2[1565] = {X 325.0031, Y 85.8502, Z -2.1667, A 0.000, B 0.000, C 0.000 }
gfCNCPoint2[1566] = {X 325.2261, Y 87.0677, Z -2.1667, A 0.000, B 0.000, C 0.000 }
gfCNCPoint2[1567] = {X 325.4715, Y 87.3367, Z -2.1667, A 0.000, B 0.000, C 0.000 }
gfCNCPoint2[1568] = {X 325.7737, Y 87.5399, Z -2.1667, A 0.000, B 0.000, C 0.000 }
gfCNCPoint2[1569] = {X 326.2236, Y 87.7937, Z -2.1667, A 0.000, B 0.000, C 0.000 }
gfCNCPoint2[1570] = {X 327.6617, Y 88.3913, Z -2.1667, A 0.000, B 0.000, C 0.000 }
gfCNCPoint2[1571] = {X 329.1568, Y 88.8270, Z -2.1667, A 0.000, B 0.000, C 0.000 }
gfCNCPoint2[1572] = {X 332.2328, Y 89.4429, Z -2.1667, A 0.000, B 0.000, C 0.000 }
gfCNCPoint2[1573] = {X 335.3452, Y 89.8353, Z -2.1667, A 0.000, B 0.000, C 0.000 }
gfCNCPoint2[1574] = {X 339.4835, Y 90.1545, Z -2.1667, A 0.000, B 0.000, C 0.000 }
gfCNCPoint2[1575] = {X 343.6301, Y 90.3342, Z -2.1667, A 0.000, B 0.000, C 0.000 }
gfCNCPoint2[1576] = {X 347.7804, Y 90.3744, Z -2.1667, A 0.000, B 0.000, C 0.000 }
gfCNCPoint2[1577] = {X 352.1621, Y 90.3360, Z -2.1667, A 0.000, B 0.000, C 0.000 }
gfCNCPoint2[1578] = {X 356.5395, Y 90.1401, Z -2.1667, A 0.000, B 0.000, C 0.000 }
gfCNCPoint2[1579] = {X 360.9071, Y 89.7870, Z -2.1667, A 0.000, B 0.000, C 0.000 }
gfCNCPoint2[1580] = {X 363.2212, Y 89.4992, Z -2.1667, A 0.000, B 0.000, C 0.000 }
gfCNCPoint2[1581] = {X 365.5139, Y 89.0729, Z -2.1667, A 0.000, B 0.000, C 0.000 }
gfCNCPoint2[1582] = {X 367.7768, Y 88.5095, Z -2.1667, A 0.000, B 0.000, C 0.000 }
gfCNCPoint2[1583] = {X 368.7090, Y 88.1961, Z -2.1667, A 0.000, B 0.000, C 0.000 }
gfCNCPoint2[1584] = {X 369.6001, Y 87.7802, Z -2.1667, A 0.000, B 0.000, C 0.000 }
gfCNCPoint2[1585] = {X 370.4390, Y 87.2669, Z -2.1667, A 0.000, B 0.000, C 0.000 }
gfCNCPoint2[1586] = {X 370.5889, Y 87.1108, Z -2.1667, A 0.000, B 0.000, C 0.000 }
gfCNCPoint2[1587] = {X 370.6662, Y 86.9086, Z -2.1667, A 0.000, B 0.000, C 0.000 }
gfCNCPoint2[1588] = {X 370.8573, Y 85.3735, Z -2.1667, A 0.000, B 0.000, C 0.000 }
gfCNCPoint2[1589] = {X 370.9211, Y 83.8278, Z -2.1667, A 0.000, B 0.000, C 0.000 }
gfCNCPoint2[1590] = {X 370.9210, Y 63.2124, Z -2.1667, A 0.000, B 0.000, C 0.000 }
gfCNCPoint2[1591] = {X 370.0692, Y 63.0034, Z -2.1667, A 0.000, B 0.000, C 0.000 }
gfCNCPoint2[1592] = {X 369.2772, Y 62.6267, Z -2.1667, A 0.000, B 0.000, C 0.000 }
gfCNCPoint2[1593] = {X 368.5776, Y 62.0977, Z -2.1667, A 0.000, B 0.000, C 0.000 }
gfCNCPoint2[1594] = {X 367.9992, Y 61.4384, Z -2.1667, A 0.000, B 0.000, C 0.000 }
gfCNCPoint2[1595] = {X 367.5660, Y 60.6758, Z -2.1667, A 0.000, B 0.000, C 0.000 }
gfCNCPoint2[1596] = {X 367.2957, Y 59.8415, Z -2.1667, A 0.000, B 0.000, C 0.000 }
gfCNCPoint2[1597] = {X 367.1994, Y 58.9697, Z -2.1667, A 0.000, B 0.000, C 0.000 }
gfCNCPoint2[1598] = {X 367.1993, Y 58.0000, Z -2.1667, A 0.000, B 0.000, C 0.000 }
gfCNCPoint2[1599] = {X 367.3076, Y 57.0387, Z -2.1667, A 0.000, B 0.000, C 0.000 }
gfCNCPoint2[1600] = {X 367.6271, Y 56.1256, Z -2.1667, A 0.000, B 0.000, C 0.000 }
gfCNCPoint2[1601] = {X 368.1418, Y 55.3065, Z -2.1667, A 0.000, B 0.000, C 0.000 }
gfCNCPoint2[1602] = {X 368.8258, Y 54.6225, Z -2.1667, A 0.000, B 0.000, C 0.000 }
gfCNCPoint2[1603] = {X 369.6449, Y 54.1078, Z -2.1667, A 0.000, B 0.000, C 0.000 }
gfCNCPoint2[1604] = {X 370.5580, Y 53.7883, Z -2.1667, A 0.000, B 0.000, C 0.000 }
gfCNCPoint2[1605] = {X 371.5193, Y 53.6800, Z -2.1667, A 0.000, B 0.000, C 0.000 }
gfCNCPoint2[1606] = {X 388.0597, Y 53.6800, Z -2.1667, A 0.000, B 0.000, C 0.000 }
gfCNCPoint2[1607] = {X 389.0210, Y 53.7883, Z -2.1667, A 0.000, B 0.000, C 0.000 }
gfCNCPoint2[1608] = {X 389.9341, Y 54.1078, Z -2.1667, A 0.000, B 0.000, C 0.000 }
gfCNCPoint2[1609] = {X 390.7532, Y 54.6225, Z -2.1667, A 0.000, B 0.000, C 0.000 }
gfCNCPoint2[1610] = {X 391.4372, Y 55.3065, Z -2.1667, A 0.000, B 0.000, C 0.000 }
gfCNCPoint2[1611] = {X 391.9519, Y 56.1256, Z -2.1667, A 0.000, B 0.000, C 0.000 }
gfCNCPoint2[1612] = {X 392.2714, Y 57.0387, Z -2.1667, A 0.000, B 0.000, C 0.000 }
gfCNCPoint2[1613] = {X 392.3797, Y 58.0000, Z -2.1667, A 0.000, B 0.000, C 0.000 }
gfCNCPoint2[1614] = {X 392.3797, Y 58.9342, Z -2.1667, A 0.000, B 0.000, C 0.000 }
gfCNCPoint2[1615] = {X 392.2641, Y 59.9267, Z -2.1667, A 0.000, B 0.000, C 0.000 }
gfCNCPoint2[1616] = {X 391.9236, Y 60.8661, Z -2.1667, A 0.000, B 0.000, C 0.000 }
gfCNCPoint2[1617] = {X 391.4799, Y 61.5754, Z -2.1667, A 0.000, B 0.000, C 0.000 }
gfCNCPoint2[1618] = {X 390.9084, Y 62.1865, Z -2.1667, A 0.000, B 0.000, C 0.000 }
gfCNCPoint2[1619] = {X 390.2303, Y 62.6765, Z -2.1667, A 0.000, B 0.000, C 0.000 }
gfCNCPoint2[1620] = {X 389.4707, Y 63.0274, Z -2.1667, A 0.000, B 0.000, C 0.000 }
gfCNCPoint2[1621] = {X 388.6580, Y 63.2260, Z -2.1667, A 0.000, B 0.000, C 0.000 }
gfCNCPoint2[1622] = {X 388.6559, Y 84.6147, Z -2.1667, A 0.000, B 0.000, C 0.000 }
gfCNCPoint2[1623] = {X 388.5957, Y 86.2730, Z -2.1667, A 0.000, B 0.000, C 0.000 }
gfCNCPoint2[1624] = {X 388.3914, Y 87.9197, Z -2.1667, A 0.000, B 0.000, C 0.000 }
gfCNCPoint2[1625] = {X 388.0445, Y 89.5424, Z -2.1667, A 0.000, B 0.000, C 0.000 }
gfCNCPoint2[1626] = {X 387.5125, Y 91.1298, Z -2.1667, A 0.000, B 0.000, C 0.000 }
gfCNCPoint2[1627] = {X 386.7629, Y 92.6269, Z -2.1667, A 0.000, B 0.000, C 0.000 }
gfCNCPoint2[1628] = {X 385.8108, Y 94.0039, Z -2.1667, A 0.000, B 0.000, C 0.000 }
gfCNCPoint2[1629] = {X 384.6748, Y 95.2338, Z -2.1667, A 0.000, B 0.000, C 0.000 }
gfCNCPoint2[1630] = {X 383.1606, Y 96.5094, Z -2.1667, A 0.000, B 0.000, C 0.000 }
gfCNCPoint2[1631] = {X 381.5196, Y 97.6172, Z -2.1667, A 0.000, B 0.000, C 0.000 }
gfCNCPoint2[1632] = {X 379.7704, Y 98.5446, Z -2.1667, A 0.000, B 0.000, C 0.000 }
gfCNCPoint2[1633] = {X 377.4992, Y 99.5007, Z -2.1667, A 0.000, B 0.000, C 0.000 }
gfCNCPoint2[1634] = {X 375.1651, Y 100.2910, Z -2.1667, A 0.000, B 0.000, C 0.000 }
gfCNCPoint2[1635] = {X 372.7802, Y 100.9113, Z -2.1667, A 0.000, B 0.000, C 0.000 }
gfCNCPoint2[1636] = {X 368.9685, Y 101.6487, Z -2.1667, A 0.000, B 0.000, C 0.000 }
gfCNCPoint2[1637] = {X 365.1257, Y 102.2021, Z -2.1667, A 0.000, B 0.000, C 0.000 }
gfCNCPoint2[1638] = {X 361.2608, Y 102.5700, Z -2.1667, A 0.000, B 0.000, C 0.000 }
gfCNCPoint2[1639] = {X 357.2538, Y 102.8107, Z -2.1667, A 0.000, B 0.000, C 0.000 }
gfCNCPoint2[1640] = {X 353.2424, Y 102.9642, Z -2.1667, A 0.000, B 0.000, C 0.000 }
gfCNCPoint2[1641] = {X 353.3519, Y 106.9627, Z -2.1667, A 0.000, B 0.000, C 0.000 }
gfCNCPoint2[1642] = {X 353.2402, Y 102.8842, Z -2.1667, A 0.000, B 0.000, C 0.000 }
gfCNCPoint2[1643] = {X 347.7204, Y 102.9527, Z -2.1667, A 0.000, B 0.000, C 0.000 }
gfCNCPoint2[1644] = {X 342.2010, Y 102.8560, Z -2.1667, A 0.000, B 0.000, C 0.000 }
gfCNCPoint2[1645] = {X 336.6869, Y 102.5942, Z -2.1667, A 0.000, B 0.000, C 0.000 }
gfCNCPoint2[1646] = {X 333.2000, Y 102.3195, Z -2.1667, A 0.000, B 0.000, C 0.000 }
gfCNCPoint2[1647] = {X 329.7268, Y 101.9069, Z -2.1667, A 0.000, B 0.000, C 0.000 }
gfCNCPoint2[1648] = {X 326.2726, Y 101.3572, Z -2.1667, A 0.000, B 0.000, C 0.000 }
gfCNCPoint2[1649] = {X 323.4288, Y 100.7537, Z -2.1667, A 0.000, B 0.000, C 0.000 }
gfCNCPoint2[1650] = {X 320.6371, Y 99.9424, Z -2.1667, A 0.000, B 0.000, C 0.000 }
gfCNCPoint2[1651] = {X 317.9128, Y 98.9277, Z -2.1667, A 0.000, B 0.000, C 0.000 }
gfCNCPoint2[1652] = {X 316.4062, Y 98.2323, Z -2.1667, A 0.000, B 0.000, C 0.000 }
gfCNCPoint2[1653] = {X 314.9629, Y 97.4136, Z -2.1667, A 0.000, B 0.000, C 0.000 }
gfCNCPoint2[1654] = {X 313.5928, Y 96.4774, Z -2.1667, A 0.000, B 0.000, C 0.000 }
gfCNCPoint2[1655] = {X 312.3057, Y 95.4302, Z -2.1667, A 0.000, B 0.000, C 0.000 }
gfCNCPoint2[1656] = {X 311.3087, Y 94.4387, Z -2.1667, A 0.000, B 0.000, C 0.000 }
gfCNCPoint2[1657] = {X 310.4363, Y 93.3359, Z -2.1667, A 0.000, B 0.000, C 0.000 }
gfCNCPoint2[1658] = {X 309.7011, Y 92.1375, Z -2.1667, A 0.000, B 0.000, C 0.000 }
gfCNCPoint2[1659] = {X 309.1132, Y 90.8602, Z -2.1667, A 0.000, B 0.000, C 0.000 }
gfCNCPoint2[1660] = {X 308.6811, Y 89.5222, Z -2.1667, A 0.000, B 0.000, C 0.000 }
gfCNCPoint2[1661] = {X 308.3390, Y 87.9058, Z -2.1667, A 0.000, B 0.000, C 0.000 }
gfCNCPoint2[1662] = {X 308.1370, Y 86.2660, Z -2.1667, A 0.000, B 0.000, C 0.000 }
gfCNCPoint2[1663] = {X 308.0764, Y 84.6149, Z -2.1667, A 0.000, B 0.000, C 0.000 }
gfCNCPoint2[1664] = {X 308.0776, Y 83.2310, Z -2.1667, A 0.000, B 0.000, C 0.000 }
gfCNCPoint2[1665] = {X 308.0776, Y 63.1422, Z -2.1667, A 0.000, B 0.000, C 0.000 }
gfCNCPoint2[1666] = {X 307.2290, Y 62.9476, Z -2.1667, A 0.000, B 0.000, C 0.000 }
gfCNCPoint2[1667] = {X 306.4381, Y 62.5837, Z -2.1667, A 0.000, B 0.000, C 0.000 }
gfCNCPoint2[1668] = {X 305.7381, Y 62.0660, Z -2.1667, A 0.000, B 0.000, C 0.000 }
gfCNCPoint2[1669] = {X 305.1587, Y 61.4161, Z -2.1667, A 0.000, B 0.000, C 0.000 }
gfCNCPoint2[1670] = {X 304.7241, Y 60.6617, Z -2.1667, A 0.000, B 0.000, C 0.000 }
gfCNCPoint2[1671] = {X 304.4529, Y 59.8344, Z -2.1667, A 0.000, B 0.000, C 0.000 }
gfCNCPoint2[1672] = {X 304.3564, Y 58.9691, Z -2.1667, A 0.000, B 0.000, C 0.000 }
gfCNCPoint2[1673] = {X 304.3562, Y 58.0000, Z -2.1667, A 0.000, B 0.000, C 0.000 }
gfCNCPoint2[1674] = {X 304.4625, Y 57.0565, Z -2.1667, A 0.000, B 0.000, C 0.000 }
gfCNCPoint2[1675] = {X 304.7761, Y 56.1603, Z -2.1667, A 0.000, B 0.000, C 0.000 }
gfCNCPoint2[1676] = {X 305.2813, Y 55.3564, Z -2.1667, A 0.000, B 0.000, C 0.000 }
gfCNCPoint2[1677] = {X 305.9526, Y 54.6850, Z -2.1667, A 0.000, B 0.000, C 0.000 }
gfCNCPoint2[1678] = {X 306.7566, Y 54.1799, Z -2.1667, A 0.000, B 0.000, C 0.000 }
gfCNCPoint2[1679] = {X 307.6527, Y 53.8663, Z -2.1667, A 0.000, B 0.000, C 0.000 }
gfCNCPoint2[1680] = {X 308.5962, Y 53.7600, Z -2.1667, A 0.000, B 0.000, C 0.000 }
gfCNCPoint2[1681] = {X 324.3107, Y 53.7600, Z -2.1667, A 0.000, B 0.000, C 0.000 }
gfCNCPoint2[1682] = {X 325.2542, Y 53.8663, Z -2.1667, A 0.000, B 0.000, C 0.000 }
gfCNCPoint2[1683] = {X 326.1504, Y 54.1799, Z -2.1667, A 0.000, B 0.000, C 0.000 }
gfCNCPoint2[1684] = {X 326.9543, Y 54.6850, Z -2.1667, A 0.000, B 0.000, C 0.000 }
gfCNCPoint2[1685] = {X 327.6257, Y 55.3564, Z -2.1667, A 0.000, B 0.000, C 0.000 }
gfCNCPoint2[1686] = {X 328.1308, Y 56.1603, Z -2.1667, A 0.000, B 0.000, C 0.000 }
gfCNCPoint2[1687] = {X 328.4444, Y 57.0565, Z -2.1667, A 0.000, B 0.000, C 0.000 }
gfCNCPoint2[1688] = {X 328.5507, Y 58.0000, Z -2.1667, A 0.000, B 0.000, C 0.000 }
gfCNCPoint2[1689] = {X 328.5507, Y 58.9356, Z -2.1667, A 0.000, B 0.000, C 0.000 }
gfCNCPoint2[1690] = {X 328.4559, Y 59.8053, Z -2.1667, A 0.000, B 0.000, C 0.000 }
gfCNCPoint2[1691] = {X 328.1862, Y 60.6376, Z -2.1667, A 0.000, B 0.000, C 0.000 }
gfCNCPoint2[1692] = {X 327.7530, Y 61.3976, Z -2.1667, A 0.000, B 0.000, C 0.000 }
gfCNCPoint2[1693] = {X 327.1742, Y 62.0537, Z -2.1667, A 0.000, B 0.000, C 0.000 }
gfCNCPoint2[1694] = {X 326.4741, Y 62.5783, Z -2.1667, A 0.000, B 0.000, C 0.000 }
gfCNCPoint2[1695] = {X 325.6819, Y 62.9496, Z -2.1667, A 0.000, B 0.000, C 0.000 }
gfCNCPoint2[1696] = {X 324.8308, Y 63.1521, Z -2.1667, A 0.000, B 0.000, C 0.000 }
gfCNCPoint2[1697] = {X 324.8322, Y 83.2300, Z -2.1667, A 0.000, B 0.000, C 0.000 }
gfCNCPoint2[1698] = {X 324.8458, Y 84.6151, Z -2.1667, A 0.000, B 0.000, C 0.000 }
gfCNCPoint2[1699] = {X 324.9246, Y 85.8674, Z -2.1667, A 0.000, B 0.000, C 0.000 }
gfCNCPoint2[1700] = {X 325.1520, Y 87.1015, Z -2.1667, A 0.000, B 0.000, C 0.000 }
gfCNCPoint2[1701] = {X 325.4127, Y 87.3917, Z -2.1667, A 0.000, B 0.000, C 0.000 }
gfCNCPoint2[1702] = {X 325.7358, Y 87.6103, Z -2.1667, A 0.000, B 0.000, C 0.000 }
gfCNCPoint2[1703] = {X 326.1865, Y 87.8647, Z -2.1667, A 0.000, B 0.000, C 0.000 }
gfCNCPoint2[1704] = {X 327.6339, Y 88.4663, Z -2.1667, A 0.000, B 0.000, C 0.000 }
gfCNCPoint2[1705] = {X 329.1387, Y 88.9049, Z -2.1667, A 0.000, B 0.000, C 0.000 }
gfCNCPoint2[1706] = {X 332.2201, Y 89.5219, Z -2.1667, A 0.000, B 0.000, C 0.000 }
gfCNCPoint2[1707] = {X 335.3381, Y 89.9150, Z -2.1667, A 0.000, B 0.000, C 0.000 }
gfCNCPoint2[1708] = {X 339.4789, Y 90.2344, Z -2.1667, A 0.000, B 0.000, C 0.000 }
gfCNCPoint2[1709] = {X 343.6281, Y 90.4142, Z -2.1667, A 0.000, B 0.000, C 0.000 }
gfCNCPoint2[1710] = {X 347.7810, Y 90.4544, Z -2.1667, A 0.000, B 0.000, C 0.000 }
gfCNCPoint2[1711] = {X 352.1651, Y 90.4159, Z -2.1667, A 0.000, B 0.000, C 0.000 }
gfCNCPoint2[1712] = {X 356.5450, Y 90.2199, Z -2.1667, A 0.000, B 0.000, C 0.000 }
gfCNCPoint2[1713] = {X 360.9150, Y 89.8667, Z -2.1667, A 0.000, B 0.000, C 0.000 }
gfCNCPoint2[1714] = {X 363.2338, Y 89.5783, Z -2.1667, A 0.000, B 0.000, C 0.000 }
gfCNCPoint2[1715] = {X 365.5310, Y 89.1510, Z -2.1667, A 0.000, B 0.000, C 0.000 }
gfCNCPoint2[1716] = {X 367.7985, Y 88.5865, Z -2.1667, A 0.000, B 0.000, C 0.000 }
gfCNCPoint2[1717] = {X 368.7390, Y 88.2703, Z -2.1667, A 0.000, B 0.000, C 0.000 }
gfCNCPoint2[1718] = {X 369.6381, Y 87.8506, Z -2.1667, A 0.000, B 0.000, C 0.000 }
gfCNCPoint2[1719] = {X 370.4845, Y 87.3326, Z -2.1667, A 0.000, B 0.000, C 0.000 }
gfCNCPoint2[1720] = {X 370.6565, Y 87.1536, Z -2.1667, A 0.000, B 0.000, C 0.000 }
gfCNCPoint2[1721] = {X 370.7451, Y 86.9217, Z -2.1667, A 0.000, B 0.000, C 0.000 }
gfCNCPoint2[1722] = {X 370.9371, Y 85.3801, Z -2.1667, A 0.000, B 0.000, C 0.000 }
gfCNCPoint2[1723] = {X 371.0011, Y 83.8278, Z -2.1667, A 0.000, B 0.000, C 0.000 }
gfCNCPoint2[1724] = {X 371.0010, Y 63.1423, Z -2.1667, A 0.000, B 0.000, C 0.000 }
gfCNCPoint2[1725] = {X 370.1523, Y 62.9477, Z -2.1667, A 0.000, B 0.000, C 0.000 }
gfCNCPoint2[1726] = {X 369.3613, Y 62.5838, Z -2.1667, A 0.000, B 0.000, C 0.000 }
gfCNCPoint2[1727] = {X 368.6613, Y 62.0661, Z -2.1667, A 0.000, B 0.000, C 0.000 }
gfCNCPoint2[1728] = {X 368.0818, Y 61.4162, Z -2.1667, A 0.000, B 0.000, C 0.000 }
gfCNCPoint2[1729] = {X 367.6472, Y 60.6617, Z -2.1667, A 0.000, B 0.000, C 0.000 }
gfCNCPoint2[1730] = {X 367.3760, Y 59.8344, Z -2.1667, A 0.000, B 0.000, C 0.000 }
gfCNCPoint2[1731] = {X 367.2794, Y 58.9691, Z -2.1667, A 0.000, B 0.000, C 0.000 }
gfCNCPoint2[1732] = {X 367.2793, Y 58.0000, Z -2.1667, A 0.000, B 0.000, C 0.000 }
gfCNCPoint2[1733] = {X 367.3856, Y 57.0565, Z -2.1667, A 0.000, B 0.000, C 0.000 }
gfCNCPoint2[1734] = {X 367.6992, Y 56.1603, Z -2.1667, A 0.000, B 0.000, C 0.000 }
gfCNCPoint2[1735] = {X 368.2043, Y 55.3564, Z -2.1667, A 0.000, B 0.000, C 0.000 }
gfCNCPoint2[1736] = {X 368.8757, Y 54.6850, Z -2.1667, A 0.000, B 0.000, C 0.000 }
gfCNCPoint2[1737] = {X 369.6796, Y 54.1799, Z -2.1667, A 0.000, B 0.000, C 0.000 }
gfCNCPoint2[1738] = {X 370.5758, Y 53.8663, Z -2.1667, A 0.000, B 0.000, C 0.000 }
gfCNCPoint2[1739] = {X 371.5193, Y 53.7600, Z -2.1667, A 0.000, B 0.000, C 0.000 }
gfCNCPoint2[1740] = {X 388.0597, Y 53.7600, Z -2.1667, A 0.000, B 0.000, C 0.000 }
gfCNCPoint2[1741] = {X 389.0032, Y 53.8663, Z -2.1667, A 0.000, B 0.000, C 0.000 }
gfCNCPoint2[1742] = {X 389.8993, Y 54.1799, Z -2.1667, A 0.000, B 0.000, C 0.000 }
gfCNCPoint2[1743] = {X 390.7033, Y 54.6850, Z -2.1667, A 0.000, B 0.000, C 0.000 }
gfCNCPoint2[1744] = {X 391.3746, Y 55.3564, Z -2.1667, A 0.000, B 0.000, C 0.000 }
gfCNCPoint2[1745] = {X 391.8798, Y 56.1603, Z -2.1667, A 0.000, B 0.000, C 0.000 }
gfCNCPoint2[1746] = {X 392.1934, Y 57.0565, Z -2.1667, A 0.000, B 0.000, C 0.000 }
gfCNCPoint2[1747] = {X 392.2997, Y 58.0000, Z -2.1667, A 0.000, B 0.000, C 0.000 }
gfCNCPoint2[1748] = {X 392.2997, Y 58.9342, Z -2.1667, A 0.000, B 0.000, C 0.000 }
gfCNCPoint2[1749] = {X 392.1862, Y 59.9083, Z -2.1667, A 0.000, B 0.000, C 0.000 }
gfCNCPoint2[1750] = {X 391.8520, Y 60.8303, Z -2.1667, A 0.000, B 0.000, C 0.000 }
gfCNCPoint2[1751] = {X 391.4081, Y 61.5375, Z -2.1667, A 0.000, B 0.000, C 0.000 }
gfCNCPoint2[1752] = {X 390.8347, Y 62.1446, Z -2.1667, A 0.000, B 0.000, C 0.000 }
gfCNCPoint2[1753] = {X 390.1540, Y 62.6282, Z -2.1667, A 0.000, B 0.000, C 0.000 }
gfCNCPoint2[1754] = {X 389.3920, Y 62.9698, Z -2.1667, A 0.000, B 0.000, C 0.000 }
gfCNCPoint2[1755] = {X 388.5780, Y 63.1562, Z -2.1667, A 0.000, B 0.000, C 0.000 }
gfCNCPoint2[1756] = {X 388.5759, Y 84.6151, Z -2.1667, A 0.000, B 0.000, C 0.000 }
gfCNCPoint2[1757] = {X 388.5160, Y 86.2665, Z -2.1667, A 0.000, B 0.000, C 0.000 }
gfCNCPoint2[1758] = {X 388.3125, Y 87.9064, Z -2.1667, A 0.000, B 0.000, C 0.000 }
gfCNCPoint2[1759] = {X 387.9671, Y 89.5224, Z -2.1667, A 0.000, B 0.000, C 0.000 }
gfCNCPoint2[1760] = {X 387.4386, Y 91.0991, Z -2.1667, A 0.000, B 0.000, C 0.000 }
gfCNCPoint2[1761] = {X 386.6941, Y 92.5861, Z -2.1667, A 0.000, B 0.000, C 0.000 }
gfCNCPoint2[1762] = {X 385.7483, Y 93.9539, Z -2.1667, A 0.000, B 0.000, C 0.000 }
gfCNCPoint2[1763] = {X 384.6200, Y 95.1755, Z -2.1667, A 0.000, B 0.000, C 0.000 }
gfCNCPoint2[1764] = {X 383.1123, Y 96.4456, Z -2.1667, A 0.000, B 0.000, C 0.000 }
gfCNCPoint2[1765] = {X 381.4784, Y 97.5486, Z -2.1667, A 0.000, B 0.000, C 0.000 }
gfCNCPoint2[1766] = {X 379.7367, Y 98.4720, Z -2.1667, A 0.000, B 0.000, C 0.000 }
gfCNCPoint2[1767] = {X 377.4708, Y 99.4259, Z -2.1667, A 0.000, B 0.000, C 0.000 }
gfCNCPoint2[1768] = {X 375.1422, Y 100.2143, Z -2.1667, A 0.000, B 0.000, C 0.000 }
gfCNCPoint2[1769] = {X 372.7628, Y 100.8332, Z -2.1667, A 0.000, B 0.000, C 0.000 }
gfCNCPoint2[1770] = {X 368.9550, Y 101.5699, Z -2.1667, A 0.000, B 0.000, C 0.000 }
gfCNCPoint2[1771] = {X 365.1161, Y 102.1227, Z -2.1667, A 0.000, B 0.000, C 0.000 }
gfCNCPoint2[1772] = {X 361.2551, Y 102.4902, Z -2.1667, A 0.000, B 0.000, C 0.000 }
gfCNCPoint2[1773] = {X 357.2498, Y 102.7308, Z -2.1667, A 0.000, B 0.000, C 0.000 }
gfCNCPoint2[1774] = {X 353.2402, Y 102.8842, Z -2.1667, A 0.000, B 0.000, C 0.000 }
gfCNCPoint2[1775] = {X 353.3497, Y 106.8827, Z -2.1667, A 0.000, B 0.000, C 0.000 }
gfCNCPoint2[1776] = {X 353.2380, Y 102.8043, Z -2.1667, A 0.000, B 0.000, C 0.000 }
gfCNCPoint2[1777] = {X 347.7206, Y 102.8727, Z -2.1667, A 0.000, B 0.000, C 0.000 }
gfCNCPoint2[1778] = {X 342.2035, Y 102.7761, Z -2.1667, A 0.000, B 0.000, C 0.000 }
gfCNCPoint2[1779] = {X 336.6918, Y 102.5144, Z -2.1667, A 0.000, B 0.000, C 0.000 }
gfCNCPoint2[1780] = {X 333.2080, Y 102.2399, Z -2.1667, A 0.000, B 0.000, C 0.000 }
gfCNCPoint2[1781] = {X 329.7377, Y 101.8277, Z -2.1667, A 0.000, B 0.000, C 0.000 }
gfCNCPoint2[1782] = {X 326.2865, Y 101.2784, Z -2.1667, A 0.000, B 0.000, C 0.000 }
gfCNCPoint2[1783] = {X 323.4484, Y 100.6761, Z -2.1667, A 0.000, B 0.000, C 0.000 }
gfCNCPoint2[1784] = {X 320.6623, Y 99.8665, Z -2.1667, A 0.000, B 0.000, C 0.000 }
gfCNCPoint2[1785] = {X 317.9434, Y 98.8538, Z -2.1667, A 0.000, B 0.000, C 0.000 }
gfCNCPoint2[1786] = {X 316.4428, Y 98.1612, Z -2.1667, A 0.000, B 0.000, C 0.000 }
gfCNCPoint2[1787] = {X 315.0052, Y 97.3458, Z -2.1667, A 0.000, B 0.000, C 0.000 }
gfCNCPoint2[1788] = {X 313.6407, Y 96.4133, Z -2.1667, A 0.000, B 0.000, C 0.000 }
gfCNCPoint2[1789] = {X 312.3587, Y 95.3703, Z -2.1667, A 0.000, B 0.000, C 0.000 }
gfCNCPoint2[1790] = {X 311.3684, Y 94.3855, Z -2.1667, A 0.000, B 0.000, C 0.000 }
gfCNCPoint2[1791] = {X 310.5020, Y 93.2902, Z -2.1667, A 0.000, B 0.000, C 0.000 }
gfCNCPoint2[1792] = {X 309.7716, Y 92.0998, Z -2.1667, A 0.000, B 0.000, C 0.000 }
gfCNCPoint2[1793] = {X 309.1877, Y 90.8311, Z -2.1667, A 0.000, B 0.000, C 0.000 }
gfCNCPoint2[1794] = {X 308.7585, Y 89.5022, Z -2.1667, A 0.000, B 0.000, C 0.000 }
gfCNCPoint2[1795] = {X 308.4179, Y 87.8924, Z -2.1667, A 0.000, B 0.000, C 0.000 }
gfCNCPoint2[1796] = {X 308.2167, Y 86.2594, Z -2.1667, A 0.000, B 0.000, C 0.000 }
gfCNCPoint2[1797] = {X 308.1564, Y 84.6152, Z -2.1667, A 0.000, B 0.000, C 0.000 }
gfCNCPoint2[1798] = {X 308.1576, Y 83.2311, Z -2.1667, A 0.000, B 0.000, C 0.000 }
gfCNCPoint2[1799] = {X 308.1576, Y 63.0709, Z -2.1667, A 0.000, B 0.000, C 0.000 }
gfCNCPoint2[1800] = {X 307.3123, Y 62.8910, Z -2.1667, A 0.000, B 0.000, C 0.000 }
gfCNCPoint2[1801] = {X 306.5224, Y 62.5403, Z -2.1667, A 0.000, B 0.000, C 0.000 }
gfCNCPoint2[1802] = {X 305.8220, Y 62.0339, Z -2.1667, A 0.000, B 0.000, C 0.000 }
gfCNCPoint2[1803] = {X 305.2413, Y 61.3938, Z -2.1667, A 0.000, B 0.000, C 0.000 }
gfCNCPoint2[1804] = {X 304.8055, Y 60.6475, Z -2.1667, A 0.000, B 0.000, C 0.000 }
gfCNCPoint2[1805] = {X 304.5332, Y 59.8272, Z -2.1667, A 0.000, B 0.000, C 0.000 }
gfCNCPoint2[1806] = {X 304.4364, Y 58.9684, Z -2.1667, A 0.000, B 0.000, C 0.000 }
gfCNCPoint2[1807] = {X 304.4362, Y 58.0000, Z -2.1667, A 0.000, B 0.000, C 0.000 }
gfCNCPoint2[1808] = {X 304.5405, Y 57.0743, Z -2.1667, A 0.000, B 0.000, C 0.000 }
gfCNCPoint2[1809] = {X 304.8482, Y 56.1950, Z -2.1667, A 0.000, B 0.000, C 0.000 }
gfCNCPoint2[1810] = {X 305.3438, Y 55.4063, Z -2.1667, A 0.000, B 0.000, C 0.000 }
gfCNCPoint2[1811] = {X 306.0025, Y 54.7476, Z -2.1667, A 0.000, B 0.000, C 0.000 }
gfCNCPoint2[1812] = {X 306.7913, Y 54.2520, Z -2.1667, A 0.000, B 0.000, C 0.000 }
gfCNCPoint2[1813] = {X 307.6705, Y 53.9443, Z -2.1667, A 0.000, B 0.000, C 0.000 }
gfCNCPoint2[1814] = {X 308.5962, Y 53.8400, Z -2.1667, A 0.000, B 0.000, C 0.000 }
gfCNCPoint2[1815] = {X 324.3107, Y 53.8400, Z -2.1667, A 0.000, B 0.000, C 0.000 }
gfCNCPoint2[1816] = {X 325.2364, Y 53.9443, Z -2.1667, A 0.000, B 0.000, C 0.000 }
gfCNCPoint2[1817] = {X 326.1156, Y 54.2520, Z -2.1667, A 0.000, B 0.000, C 0.000 }
gfCNCPoint2[1818] = {X 326.9044, Y 54.7476, Z -2.1667, A 0.000, B 0.000, C 0.000 }
gfCNCPoint2[1819] = {X 327.5631, Y 55.4063, Z -2.1667, A 0.000, B 0.000, C 0.000 }
gfCNCPoint2[1820] = {X 328.0587, Y 56.1950, Z -2.1667, A 0.000, B 0.000, C 0.000 }
gfCNCPoint2[1821] = {X 328.3664, Y 57.0743, Z -2.1667, A 0.000, B 0.000, C 0.000 }
gfCNCPoint2[1822] = {X 328.4707, Y 58.0000, Z -2.1667, A 0.000, B 0.000, C 0.000 }
gfCNCPoint2[1823] = {X 328.4707, Y 58.9351, Z -2.1667, A 0.000, B 0.000, C 0.000 }
gfCNCPoint2[1824] = {X 328.3756, Y 59.7983, Z -2.1667, A 0.000, B 0.000, C 0.000 }
gfCNCPoint2[1825] = {X 328.1049, Y 60.6236, Z -2.1667, A 0.000, B 0.000, C 0.000 }
gfCNCPoint2[1826] = {X 327.6703, Y 61.3755, Z -2.1667, A 0.000, B 0.000, C 0.000 }
gfCNCPoint2[1827] = {X 327.0904, Y 62.0219, Z -2.1667, A 0.000, B 0.000, C 0.000 }
gfCNCPoint2[1828] = {X 326.3898, Y 62.5352, Z -2.1667, A 0.000, B 0.000, C 0.000 }
gfCNCPoint2[1829] = {X 325.5987, Y 62.8935, Z -2.1667, A 0.000, B 0.000, C 0.000 }
gfCNCPoint2[1830] = {X 324.7508, Y 63.0814, Z -2.1667, A 0.000, B 0.000, C 0.000 }
gfCNCPoint2[1831] = {X 324.7522, Y 83.2304, Z -2.1667, A 0.000, B 0.000, C 0.000 }
gfCNCPoint2[1832] = {X 324.7658, Y 84.6154, Z -2.1667, A 0.000, B 0.000, C 0.000 }
gfCNCPoint2[1833] = {X 324.8461, Y 85.8845, Z -2.1667, A 0.000, B 0.000, C 0.000 }
gfCNCPoint2[1834] = {X 325.0778, Y 87.1349, Z -2.1667, A 0.000, B 0.000, C 0.000 }
gfCNCPoint2[1835] = {X 325.3539, Y 87.4465, Z -2.1667, A 0.000, B 0.000, C 0.000 }
gfCNCPoint2[1836] = {X 325.6979, Y 87.6808, Z -2.1667, A 0.000, B 0.000, C 0.000 }
gfCNCPoint2[1837] = {X 326.1494, Y 87.9356, Z -2.1667, A 0.000, B 0.000, C 0.000 }
gfCNCPoint2[1838] = {X 327.6060, Y 88.5414, Z -2.1667, A 0.000, B 0.000, C 0.000 }
gfCNCPoint2[1839] = {X 329.1206, Y 88.9828, Z -2.1667, A 0.000, B 0.000, C 0.000 }
gfCNCPoint2[1840] = {X 332.2075, Y 89.6008, Z -2.1667, A 0.000, B 0.000, C 0.000 }
gfCNCPoint2[1841] = {X 335.3310, Y 89.9947, Z -2.1667, A 0.000, B 0.000, C 0.000 }
gfCNCPoint2[1842] = {X 339.4743, Y 90.3142, Z -2.1667, A 0.000, B 0.000, C 0.000 }
gfCNCPoint2[1843] = {X 343.6261, Y 90.4942, Z -2.1667, A 0.000, B 0.000, C 0.000 }
gfCNCPoint2[1844] = {X 347.7816, Y 90.5344, Z -2.1667, A 0.000, B 0.000, C 0.000 }
gfCNCPoint2[1845] = {X 352.1681, Y 90.4959, Z -2.1667, A 0.000, B 0.000, C 0.000 }
gfCNCPoint2[1846] = {X 356.5504, Y 90.2997, Z -2.1667, A 0.000, B 0.000, C 0.000 }
gfCNCPoint2[1847] = {X 360.9228, Y 89.9463, Z -2.1667, A 0.000, B 0.000, C 0.000 }
gfCNCPoint2[1848] = {X 363.2463, Y 89.6573, Z -2.1667, A 0.000, B 0.000, C 0.000 }
gfCNCPoint2[1849] = {X 365.5481, Y 89.2292, Z -2.1667, A 0.000, B 0.000, C 0.000 }
gfCNCPoint2[1850] = {X 367.8201, Y 88.6635, Z -2.1667, A 0.000, B 0.000, C 0.000 }
gfCNCPoint2[1851] = {X 368.7690, Y 88.3444, Z -2.1667, A 0.000, B 0.000, C 0.000 }
gfCNCPoint2[1852] = {X 369.6761, Y 87.9210, Z -2.1667, A 0.000, B 0.000, C 0.000 }
gfCNCPoint2[1853] = {X 370.5300, Y 87.3984, Z -2.1667, A 0.000, B 0.000, C 0.000 }
gfCNCPoint2[1854] = {X 370.7240, Y 87.1965, Z -2.1667, A 0.000, B 0.000, C 0.000 }
gfCNCPoint2[1855] = {X 370.8241, Y 86.9349, Z -2.1667, A 0.000, B 0.000, C 0.000 }
gfCNCPoint2[1856] = {X 371.0168, Y 85.3866, Z -2.1667, A 0.000, B 0.000, C 0.000 }
gfCNCPoint2[1857] = {X 371.0811, Y 83.8278, Z -2.1667, A 0.000, B 0.000, C 0.000 }
gfCNCPoint2[1858] = {X 371.0810, Y 63.0709, Z -2.1667, A 0.000, B 0.000, C 0.000 }
gfCNCPoint2[1859] = {X 370.9786, Y 63.0588, Z -2.1667, A 0.000, B 0.000, C 0.000 }
gfCNCPoint2[1860] = {X 370.8765, Y 63.0441, Z -2.1667, A 0.000, B 0.000, C 0.000 }
gfCNCPoint2[1861] = {X 369.9388, Y 62.7822, Z -2.1667, A 0.000, B 0.000, C 0.000 }
gfCNCPoint2[1862] = {X 369.0877, Y 62.3094, Z -2.1667, A 0.000, B 0.000, C 0.000 }
gfCNCPoint2[1863] = {X 368.3698, Y 61.6519, Z -2.1667, A 0.000, B 0.000, C 0.000 }
gfCNCPoint2[1864] = {X 367.8244, Y 60.8454, Z -2.1667, A 0.000, B 0.000, C 0.000 }
gfCNCPoint2[1865] = {X 367.4813, Y 59.9343, Z -2.1667, A 0.000, B 0.000, C 0.000 }
gfCNCPoint2[1866] = {X 367.3594, Y 58.9684, Z -2.1667, A 0.000, B 0.000, C 0.000 }
gfCNCPoint2[1867] = {X 367.3593, Y 58.0000, Z -2.1667, A 0.000, B 0.000, C 0.000 }
gfCNCPoint2[1868] = {X 367.4636, Y 57.0743, Z -2.1667, A 0.000, B 0.000, C 0.000 }
gfCNCPoint2[1869] = {X 367.7713, Y 56.1950, Z -2.1667, A 0.000, B 0.000, C 0.000 }
gfCNCPoint2[1870] = {X 368.2669, Y 55.4063, Z -2.1667, A 0.000, B 0.000, C 0.000 }
gfCNCPoint2[1871] = {X 368.9256, Y 54.7476, Z -2.1667, A 0.000, B 0.000, C 0.000 }
gfCNCPoint2[1872] = {X 369.7143, Y 54.2520, Z -2.1667, A 0.000, B 0.000, C 0.000 }
gfCNCPoint2[1873] = {X 370.5936, Y 53.9443, Z -2.1667, A 0.000, B 0.000, C 0.000 }
gfCNCPoint2[1874] = {X 371.5193, Y 53.8400, Z -2.1667, A 0.000, B 0.000, C 0.000 }
gfCNCPoint2[1875] = {X 388.0597, Y 53.8400, Z -2.1667, A 0.000, B 0.000, C 0.000 }
gfCNCPoint2[1876] = {X 388.9854, Y 53.9443, Z -2.1667, A 0.000, B 0.000, C 0.000 }
gfCNCPoint2[1877] = {X 389.8646, Y 54.2520, Z -2.1667, A 0.000, B 0.000, C 0.000 }
gfCNCPoint2[1878] = {X 390.6534, Y 54.7476, Z -2.1667, A 0.000, B 0.000, C 0.000 }
gfCNCPoint2[1879] = {X 391.3121, Y 55.4063, Z -2.1667, A 0.000, B 0.000, C 0.000 }
gfCNCPoint2[1880] = {X 391.8077, Y 56.1950, Z -2.1667, A 0.000, B 0.000, C 0.000 }
gfCNCPoint2[1881] = {X 392.1154, Y 57.0743, Z -2.1667, A 0.000, B 0.000, C 0.000 }
gfCNCPoint2[1882] = {X 392.2197, Y 58.0000, Z -2.1667, A 0.000, B 0.000, C 0.000 }
gfCNCPoint2[1883] = {X 392.2197, Y 58.9342, Z -2.1667, A 0.000, B 0.000, C 0.000 }
gfCNCPoint2[1884] = {X 392.1084, Y 59.8899, Z -2.1667, A 0.000, B 0.000, C 0.000 }
gfCNCPoint2[1885] = {X 391.7805, Y 60.7945, Z -2.1667, A 0.000, B 0.000, C 0.000 }
gfCNCPoint2[1886] = {X 391.2364, Y 61.6209, Z -2.1667, A 0.000, B 0.000, C 0.000 }
gfCNCPoint2[1887] = {X 390.5133, Y 62.2963, Z -2.1667, A 0.000, B 0.000, C 0.000 }
gfCNCPoint2[1888] = {X 389.6518, Y 62.7828, Z -2.1667, A 0.000, B 0.000, C 0.000 }
gfCNCPoint2[1889] = {X 388.7001, Y 63.0534, Z -2.1667, A 0.000, B 0.000, C 0.000 }
gfCNCPoint2[1890] = {X 388.5999, Y 63.0681, Z -2.1667, A 0.000, B 0.000, C 0.000 }
gfCNCPoint2[1891] = {X 388.4993, Y 63.0804, Z -2.1667, A 0.000, B 0.000, C 0.000 }
gfCNCPoint2[1892] = {X 388.4959, Y 84.6154, Z -2.1667, A 0.000, B 0.000, C 0.000 }
gfCNCPoint2[1893] = {X 388.4362, Y 86.2599, Z -2.1667, A 0.000, B 0.000, C 0.000 }
gfCNCPoint2[1894] = {X 388.2336, Y 87.8930, Z -2.1667, A 0.000, B 0.000, C 0.000 }
gfCNCPoint2[1895] = {X 387.8896, Y 89.5023, Z -2.1667, A 0.000, B 0.000, C 0.000 }
gfCNCPoint2[1896] = {X 387.3647, Y 91.0684, Z -2.1667, A 0.000, B 0.000, C 0.000 }
gfCNCPoint2[1897] = {X 386.6253, Y 92.5453, Z -2.1667, A 0.000, B 0.000, C 0.000 }
gfCNCPoint2[1898] = {X 385.6859, Y 93.9039, Z -2.1667, A 0.000, B 0.000, C 0.000 }
gfCNCPoint2[1899] = {X 384.5652, Y 95.1172, Z -2.1667, A 0.000, B 0.000, C 0.000 }
gfCNCPoint2[1900] = {X 383.0641, Y 96.3818, Z -2.1667, A 0.000, B 0.000, C 0.000 }
gfCNCPoint2[1901] = {X 381.4372, Y 97.4800, Z -2.1667, A 0.000, B 0.000, C 0.000 }
gfCNCPoint2[1902] = {X 379.7030, Y 98.3994, Z -2.1667, A 0.000, B 0.000, C 0.000 }
gfCNCPoint2[1903] = {X 377.4424, Y 99.3511, Z -2.1667, A 0.000, B 0.000, C 0.000 }
gfCNCPoint2[1904] = {X 375.1192, Y 100.1377, Z -2.1667, A 0.000, B 0.000, C 0.000 }
gfCNCPoint2[1905] = {X 372.7455, Y 100.7551, Z -2.1667, A 0.000, B 0.000, C 0.000 }
gfCNCPoint2[1906] = {X 368.9415, Y 101.4910, Z -2.1667, A 0.000, B 0.000, C 0.000 }
gfCNCPoint2[1907] = {X 365.1066, Y 102.0432, Z -2.1667, A 0.000, B 0.000, C 0.000 }
gfCNCPoint2[1908] = {X 361.2495, Y 102.4104, Z -2.1667, A 0.000, B 0.000, C 0.000 }
gfCNCPoint2[1909] = {X 357.2459, Y 102.6509, Z -2.1667, A 0.000, B 0.000, C 0.000 }
gfCNCPoint2[1910] = {X 353.2380, Y 102.8043, Z -2.1667, A 0.000, B 0.000, C 0.000 }
gfCNCPoint2[1911] = {X 353.3475, Y 106.8028, Z -2.1667, A 0.000, B 0.000, C 0.000 }
gfCNCPoint2[1912] = {X 353.2359, Y 102.7243, Z -2.1667, A 0.000, B 0.000, C 0.000 }
gfCNCPoint2[1913] = {X 347.7208, Y 102.7927, Z -2.1667, A 0.000, B 0.000, C 0.000 }
gfCNCPoint2[1914] = {X 342.2061, Y 102.6961, Z -2.1667, A 0.000, B 0.000, C 0.000 }
gfCNCPoint2[1915] = {X 336.6968, Y 102.4346, Z -2.1667, A 0.000, B 0.000, C 0.000 }
gfCNCPoint2[1916] = {X 333.2159, Y 102.1603, Z -2.1667, A 0.000, B 0.000, C 0.000 }
gfCNCPoint2[1917] = {X 329.7487, Y 101.7484, Z -2.1667, A 0.000, B 0.000, C 0.000 }
gfCNCPoint2[1918] = {X 326.3005, Y 101.1996, Z -2.1667, A 0.000, B 0.000, C 0.000 }
gfCNCPoint2[1919] = {X 323.4680, Y 100.5986, Z -2.1667, A 0.000, B 0.000, C 0.000 }
gfCNCPoint2[1920] = {X 320.6875, Y 99.7905, Z -2.1667, A 0.000, B 0.000, C 0.000 }
gfCNCPoint2[1921] = {X 317.9740, Y 98.7798, Z -2.1667, A 0.000, B 0.000, C 0.000 }
gfCNCPoint2[1922] = {X 316.4794, Y 98.0900, Z -2.1667, A 0.000, B 0.000, C 0.000 }
gfCNCPoint2[1923] = {X 315.0476, Y 97.2779, Z -2.1667, A 0.000, B 0.000, C 0.000 }
gfCNCPoint2[1924] = {X 313.6886, Y 96.3492, Z -2.1667, A 0.000, B 0.000, C 0.000 }
gfCNCPoint2[1925] = {X 312.4117, Y 95.3103, Z -2.1667, A 0.000, B 0.000, C 0.000 }
gfCNCPoint2[1926] = {X 311.4281, Y 94.3323, Z -2.1667, A 0.000, B 0.000, C 0.000 }
gfCNCPoint2[1927] = {X 310.5676, Y 93.2444, Z -2.1667, A 0.000, B 0.000, C 0.000 }
gfCNCPoint2[1928] = {X 309.8422, Y 92.0621, Z -2.1667, A 0.000, B 0.000, C 0.000 }
gfCNCPoint2[1929] = {X 309.2623, Y 90.8021, Z -2.1667, A 0.000, B 0.000, C 0.000 }
gfCNCPoint2[1930] = {X 308.8360, Y 89.4821, Z -2.1667, A 0.000, B 0.000, C 0.000 }
gfCNCPoint2[1931] = {X 308.4968, Y 87.8791, Z -2.1667, A 0.000, B 0.000, C 0.000 }
gfCNCPoint2[1932] = {X 308.2964, Y 86.2529, Z -2.1667, A 0.000, B 0.000, C 0.000 }
gfCNCPoint2[1933] = {X 308.2364, Y 84.6155, Z -2.1667, A 0.000, B 0.000, C 0.000 }
gfCNCPoint2[1934] = {X 308.2376, Y 83.2312, Z -2.1667, A 0.000, B 0.000, C 0.000 }
gfCNCPoint2[1935] = {X 308.2376, Y 62.9983, Z -2.1667, A 0.000, B 0.000, C 0.000 }
gfCNCPoint2[1936] = {X 307.3958, Y 62.8335, Z -2.1667, A 0.000, B 0.000, C 0.000 }
gfCNCPoint2[1937] = {X 306.6070, Y 62.4963, Z -2.1667, A 0.000, B 0.000, C 0.000 }
gfCNCPoint2[1938] = {X 305.9061, Y 62.0016, Z -2.1667, A 0.000, B 0.000, C 0.000 }
gfCNCPoint2[1939] = {X 305.3242, Y 61.3713, Z -2.1667, A 0.000, B 0.000, C 0.000 }
gfCNCPoint2[1940] = {X 304.8869, Y 60.6332, Z -2.1667, A 0.000, B 0.000, C 0.000 }
gfCNCPoint2[1941] = {X 304.6136, Y 59.8201, Z -2.1667, A 0.000, B 0.000, C 0.000 }
gfCNCPoint2[1942] = {X 304.5164, Y 58.9678, Z -2.1667, A 0.000, B 0.000, C 0.000 }
gfCNCPoint2[1943] = {X 304.5162, Y 58.0000, Z -2.1667, A 0.000, B 0.000, C 0.000 }
gfCNCPoint2[1944] = {X 304.6185, Y 57.0921, Z -2.1667, A 0.000, B 0.000, C 0.000 }
gfCNCPoint2[1945] = {X 304.9203, Y 56.2298, Z -2.1667, A 0.000, B 0.000, C 0.000 }
gfCNCPoint2[1946] = {X 305.4064, Y 55.4562, Z -2.1667, A 0.000, B 0.000, C 0.000 }
gfCNCPoint2[1947] = {X 306.0524, Y 54.8101, Z -2.1667, A 0.000, B 0.000, C 0.000 }
gfCNCPoint2[1948] = {X 306.8260, Y 54.3240, Z -2.1667, A 0.000, B 0.000, C 0.000 }
gfCNCPoint2[1949] = {X 307.6883, Y 54.0223, Z -2.1667, A 0.000, B 0.000, C 0.000 }
gfCNCPoint2[1950] = {X 308.5962, Y 53.9200, Z -2.1667, A 0.000, B 0.000, C 0.000 }
gfCNCPoint2[1951] = {X 324.3107, Y 53.9200, Z -2.1667, A 0.000, B 0.000, C 0.000 }
gfCNCPoint2[1952] = {X 325.2186, Y 54.0223, Z -2.1667, A 0.000, B 0.000, C 0.000 }
gfCNCPoint2[1953] = {X 326.0809, Y 54.3240, Z -2.1667, A 0.000, B 0.000, C 0.000 }
gfCNCPoint2[1954] = {X 326.8545, Y 54.8101, Z -2.1667, A 0.000, B 0.000, C 0.000 }
gfCNCPoint2[1955] = {X 327.5006, Y 55.4562, Z -2.1667, A 0.000, B 0.000, C 0.000 }
gfCNCPoint2[1956] = {X 327.9866, Y 56.2298, Z -2.1667, A 0.000, B 0.000, C 0.000 }
gfCNCPoint2[1957] = {X 328.2884, Y 57.0921, Z -2.1667, A 0.000, B 0.000, C 0.000 }
gfCNCPoint2[1958] = {X 328.3907, Y 58.0000, Z -2.1667, A 0.000, B 0.000, C 0.000 }
gfCNCPoint2[1959] = {X 328.3907, Y 58.9346, Z -2.1667, A 0.000, B 0.000, C 0.000 }
gfCNCPoint2[1960] = {X 328.2952, Y 59.7913, Z -2.1667, A 0.000, B 0.000, C 0.000 }
gfCNCPoint2[1961] = {X 328.0235, Y 60.6095, Z -2.1667, A 0.000, B 0.000, C 0.000 }
gfCNCPoint2[1962] = {X 327.5875, Y 61.3531, Z -2.1667, A 0.000, B 0.000, C 0.000 }
gfCNCPoint2[1963] = {X 327.0063, Y 61.9898, Z -2.1667, A 0.000, B 0.000, C 0.000 }
gfCNCPoint2[1964] = {X 326.3054, Y 62.4916, Z -2.1667, A 0.000, B 0.000, C 0.000 }
gfCNCPoint2[1965] = {X 325.5153, Y 62.8365, Z -2.1667, A 0.000, B 0.000, C 0.000 }
gfCNCPoint2[1966] = {X 324.6708, Y 63.0094, Z -2.1667, A 0.000, B 0.000, C 0.000 }
gfCNCPoint2[1967] = {X 324.6722, Y 83.2308, Z -2.1667, A 0.000, B 0.000, C 0.000 }
gfCNCPoint2[1968] = {X 324.6858, Y 84.6156, Z -2.1667, A 0.000, B 0.000, C 0.000 }
gfCNCPoint2[1969] = {X 324.7676, Y 85.9015, Z -2.1667, A 0.000, B 0.000, C 0.000 }
gfCNCPoint2[1970] = {X 325.0037, Y 87.1681, Z -2.1667, A 0.000, B 0.000, C 0.000 }
gfCNCPoint2[1971] = {X 325.2949, Y 87.5011, Z -2.1667, A 0.000, B 0.000, C 0.000 }
gfCNCPoint2[1972] = {X 325.6599, Y 87.7512, Z -2.1667, A 0.000, B 0.000, C 0.000 }
gfCNCPoint2[1973] = {X 326.1124, Y 88.0066, Z -2.1667, A 0.000, B 0.000, C 0.000 }
gfCNCPoint2[1974] = {X 327.5782, Y 88.6164, Z -2.1667, A 0.000, B 0.000, C 0.000 }
gfCNCPoint2[1975] = {X 329.1024, Y 89.0608, Z -2.1667, A 0.000, B 0.000, C 0.000 }
gfCNCPoint2[1976] = {X 332.1948, Y 89.6798, Z -2.1667, A 0.000, B 0.000, C 0.000 }
gfCNCPoint2[1977] = {X 335.3238, Y 90.0744, Z -2.1667, A 0.000, B 0.000, C 0.000 }
gfCNCPoint2[1978] = {X 339.4695, Y 90.3941, Z -2.1667, A 0.000, B 0.000, C 0.000 }
gfCNCPoint2[1979] = {X 343.6236, Y 90.5741, Z -2.1667, A 0.000, B 0.000, C 0.000 }
gfCNCPoint2[1980] = {X 347.7815, Y 90.6144, Z -2.1667, A 0.000, B 0.000, C 0.000 }
gfCNCPoint2[1981] = {X 352.1707, Y 90.5758, Z -2.1667, A 0.000, B 0.000, C 0.000 }
gfCNCPoint2[1982] = {X 356.5556, Y 90.3796, Z -2.1667, A 0.000, B 0.000, C 0.000 }
gfCNCPoint2[1983] = {X 360.9307, Y 90.0259, Z -2.1667, A 0.000, B 0.000, C 0.000 }
gfCNCPoint2[1984] = {X 363.2588, Y 89.7363, Z -2.1667, A 0.000, B 0.000, C 0.000 }
gfCNCPoint2[1985] = {X 365.5653, Y 89.3073, Z -2.1667, A 0.000, B 0.000, C 0.000 }
gfCNCPoint2[1986] = {X 367.8418, Y 88.7405, Z -2.1667, A 0.000, B 0.000, C 0.000 }
gfCNCPoint2[1987] = {X 368.7990, Y 88.4186, Z -2.1667, A 0.000, B 0.000, C 0.000 }
gfCNCPoint2[1988] = {X 369.7141, Y 87.9914, Z -2.1667, A 0.000, B 0.000, C 0.000 }
gfCNCPoint2[1989] = {X 370.5755, Y 87.4642, Z -2.1667, A 0.000, B 0.000, C 0.000 }
gfCNCPoint2[1990] = {X 370.7916, Y 87.2393, Z -2.1667, A 0.000, B 0.000, C 0.000 }
gfCNCPoint2[1991] = {X 370.9030, Y 86.9481, Z -2.1667, A 0.000, B 0.000, C 0.000 }
gfCNCPoint2[1992] = {X 371.0965, Y 85.3932, Z -2.1667, A 0.000, B 0.000, C 0.000 }
gfCNCPoint2[1993] = {X 371.1611, Y 83.8278, Z -2.1667, A 0.000, B 0.000, C 0.000 }
gfCNCPoint2[1994] = {X 371.1610, Y 62.9983, Z -2.1667, A 0.000, B 0.000, C 0.000 }
gfCNCPoint2[1995] = {X 371.0246, Y 62.9840, Z -2.1667, A 0.000, B 0.000, C 0.000 }
gfCNCPoint2[1996] = {X 370.8888, Y 62.9651, Z -2.1667, A 0.000, B 0.000, C 0.000 }
gfCNCPoint2[1997] = {X 369.9692, Y 62.7082, Z -2.1667, A 0.000, B 0.000, C 0.000 }
gfCNCPoint2[1998] = {X 369.1345, Y 62.2445, Z -2.1667, A 0.000, B 0.000, C 0.000 }
gfCNCPoint2[1999] = {X 368.4304, Y 61.5996, Z -2.1667, A 0.000, B 0.000, C 0.000 }
gfCNCPoint2[2000] = {X 367.8954, Y 60.8087, Z -2.1667, A 0.000, B 0.000, C 0.000 }
gfCNCPoint2[2001] = {X 367.5590, Y 59.9151, Z -2.1667, A 0.000, B 0.000, C 0.000 }
gfCNCPoint2[2002] = {X 367.4394, Y 58.9678, Z -2.1667, A 0.000, B 0.000, C 0.000 }
gfCNCPoint2[2003] = {X 367.4393, Y 58.0000, Z -2.1667, A 0.000, B 0.000, C 0.000 }
gfCNCPoint2[2004] = {X 367.5416, Y 57.0921, Z -2.1667, A 0.000, B 0.000, C 0.000 }
gfCNCPoint2[2005] = {X 367.8433, Y 56.2298, Z -2.1667, A 0.000, B 0.000, C 0.000 }
gfCNCPoint2[2006] = {X 368.3294, Y 55.4562, Z -2.1667, A 0.000, B 0.000, C 0.000 }
gfCNCPoint2[2007] = {X 368.9754, Y 54.8101, Z -2.1667, A 0.000, B 0.000, C 0.000 }
gfCNCPoint2[2008] = {X 369.7490, Y 54.3240, Z -2.1667, A 0.000, B 0.000, C 0.000 }
gfCNCPoint2[2009] = {X 370.6114, Y 54.0223, Z -2.1667, A 0.000, B 0.000, C 0.000 }
gfCNCPoint2[2010] = {X 371.5193, Y 53.9200, Z -2.1667, A 0.000, B 0.000, C 0.000 }
gfCNCPoint2[2011] = {X 388.0597, Y 53.9200, Z -2.1667, A 0.000, B 0.000, C 0.000 }
gfCNCPoint2[2012] = {X 388.9676, Y 54.0223, Z -2.1667, A 0.000, B 0.000, C 0.000 }
gfCNCPoint2[2013] = {X 389.8299, Y 54.3240, Z -2.1667, A 0.000, B 0.000, C 0.000 }
gfCNCPoint2[2014] = {X 390.6035, Y 54.8101, Z -2.1667, A 0.000, B 0.000, C 0.000 }
gfCNCPoint2[2015] = {X 391.2496, Y 55.4562, Z -2.1667, A 0.000, B 0.000, C 0.000 }
gfCNCPoint2[2016] = {X 391.7356, Y 56.2298, Z -2.1667, A 0.000, B 0.000, C 0.000 }
gfCNCPoint2[2017] = {X 392.0374, Y 57.0921, Z -2.1667, A 0.000, B 0.000, C 0.000 }
gfCNCPoint2[2018] = {X 392.1397, Y 58.0000, Z -2.1667, A 0.000, B 0.000, C 0.000 }
gfCNCPoint2[2019] = {X 392.1397, Y 58.9342, Z -2.1667, A 0.000, B 0.000, C 0.000 }
gfCNCPoint2[2020] = {X 392.0305, Y 59.8715, Z -2.1667, A 0.000, B 0.000, C 0.000 }
gfCNCPoint2[2021] = {X 391.7089, Y 60.7587, Z -2.1667, A 0.000, B 0.000, C 0.000 }
gfCNCPoint2[2022] = {X 391.1752, Y 61.5693, Z -2.1667, A 0.000, B 0.000, C 0.000 }
gfCNCPoint2[2023] = {X 390.4660, Y 62.2318, Z -2.1667, A 0.000, B 0.000, C 0.000 }
gfCNCPoint2[2024] = {X 389.6210, Y 62.7090, Z -2.1667, A 0.000, B 0.000, C 0.000 }
gfCNCPoint2[2025] = {X 388.6875, Y 62.9744, Z -2.1667, A 0.000, B 0.000, C 0.000 }
gfCNCPoint2[2026] = {X 388.5543, Y 62.9934, Z -2.1667, A 0.000, B 0.000, C 0.000 }
gfCNCPoint2[2027] = {X 388.4205, Y 63.0080, Z -2.1667, A 0.000, B 0.000, C 0.000 }
gfCNCPoint2[2028] = {X 388.4180, Y 63.1547, Z -2.1667, A 0.000, B 0.000, C 0.000 }
gfCNCPoint2[2029] = {X 388.4159, Y 84.6157, Z -2.1667, A 0.000, B 0.000, C 0.000 }
gfCNCPoint2[2030] = {X 388.3565, Y 86.2534, Z -2.1667, A 0.000, B 0.000, C 0.000 }
gfCNCPoint2[2031] = {X 388.1547, Y 87.8797, Z -2.1667, A 0.000, B 0.000, C 0.000 }
gfCNCPoint2[2032] = {X 387.8122, Y 89.4822, Z -2.1667, A 0.000, B 0.000, C 0.000 }
gfCNCPoint2[2033] = {X 387.2908, Y 91.0377, Z -2.1667, A 0.000, B 0.000, C 0.000 }
gfCNCPoint2[2034] = {X 386.5564, Y 92.5045, Z -2.1667, A 0.000, B 0.000, C 0.000 }
gfCNCPoint2[2035] = {X 385.6235, Y 93.8539, Z -2.1667, A 0.000, B 0.000, C 0.000 }
gfCNCPoint2[2036] = {X 384.5104, Y 95.0589, Z -2.1667, A 0.000, B 0.000, C 0.000 }
gfCNCPoint2[2037] = {X 383.0158, Y 96.3181, Z -2.1667, A 0.000, B 0.000, C 0.000 }
gfCNCPoint2[2038] = {X 381.3960, Y 97.4115, Z -2.1667, A 0.000, B 0.000, C 0.000 }
gfCNCPoint2[2039] = {X 379.6693, Y 98.3269, Z -2.1667, A 0.000, B 0.000, C 0.000 }
gfCNCPoint2[2040] = {X 377.4141, Y 99.2763, Z -2.1667, A 0.000, B 0.000, C 0.000 }
gfCNCPoint2[2041] = {X 375.0963, Y 100.0610, Z -2.1667, A 0.000, B 0.000, C 0.000 }
gfCNCPoint2[2042] = {X 372.7282, Y 100.6770, Z -2.1667, A 0.000, B 0.000, C 0.000 }
gfCNCPoint2[2043] = {X 368.9280, Y 101.4122, Z -2.1667, A 0.000, B 0.000, C 0.000 }
gfCNCPoint2[2044] = {X 365.0970, Y 101.9638, Z -2.1667, A 0.000, B 0.000, C 0.000 }
gfCNCPoint2[2045] = {X 361.2438, Y 102.3306, Z -2.1667, A 0.000, B 0.000, C 0.000 }
gfCNCPoint2[2046] = {X 357.2420, Y 102.5710, Z -2.1667, A 0.000, B 0.000, C 0.000 }
gfCNCPoint2[2047] = {X 353.2359, Y 102.7243, Z -2.1667, A 0.000, B 0.000, C 0.000 }
gfCNCPoint2[2048] = {X 353.3453, Y 106.7228, Z -2.1667, A 0.000, B 0.000, C 0.000 }
gfCNCPoint2[2049] = {X 353.2337, Y 102.6443, Z -2.1667, A 0.000, B 0.000, C 0.000 }
gfCNCPoint2[2050] = {X 347.7209, Y 102.7127, Z -2.1667, A 0.000, B 0.000, C 0.000 }
gfCNCPoint2[2051] = {X 342.2086, Y 102.6162, Z -2.1667, A 0.000, B 0.000, C 0.000 }
gfCNCPoint2[2052] = {X 336.7017, Y 102.3547, Z -2.1667, A 0.000, B 0.000, C 0.000 }
gfCNCPoint2[2053] = {X 333.2238, Y 102.0807, Z -2.1667, A 0.000, B 0.000, C 0.000 }
gfCNCPoint2[2054] = {X 329.7596, Y 101.6692, Z -2.1667, A 0.000, B 0.000, C 0.000 }
gfCNCPoint2[2055] = {X 326.3144, Y 101.1208, Z -2.1667, A 0.000, B 0.000, C 0.000 }
gfCNCPoint2[2056] = {X 323.4876, Y 100.5210, Z -2.1667, A 0.000, B 0.000, C 0.000 }
gfCNCPoint2[2057] = {X 320.7126, Y 99.7146, Z -2.1667, A 0.000, B 0.000, C 0.000 }
gfCNCPoint2[2058] = {X 318.0046, Y 98.7059, Z -2.1667, A 0.000, B 0.000, C 0.000 }
gfCNCPoint2[2059] = {X 316.5160, Y 98.0189, Z -2.1667, A 0.000, B 0.000, C 0.000 }
gfCNCPoint2[2060] = {X 315.0900, Y 97.2101, Z -2.1667, A 0.000, B 0.000, C 0.000 }
gfCNCPoint2[2061] = {X 313.7364, Y 96.2851, Z -2.1667, A 0.000, B 0.000, C 0.000 }
gfCNCPoint2[2062] = {X 312.4647, Y 95.2504, Z -2.1667, A 0.000, B 0.000, C 0.000 }
gfCNCPoint2[2063] = {X 311.4879, Y 94.2791, Z -2.1667, A 0.000, B 0.000, C 0.000 }
gfCNCPoint2[2064] = {X 310.6332, Y 93.1986, Z -2.1667, A 0.000, B 0.000, C 0.000 }
gfCNCPoint2[2065] = {X 309.9128, Y 92.0244, Z -2.1667, A 0.000, B 0.000, C 0.000 }
gfCNCPoint2[2066] = {X 309.3368, Y 90.7730, Z -2.1667, A 0.000, B 0.000, C 0.000 }
gfCNCPoint2[2067] = {X 308.9134, Y 89.4621, Z -2.1667, A 0.000, B 0.000, C 0.000 }
gfCNCPoint2[2068] = {X 308.5757, Y 87.8658, Z -2.1667, A 0.000, B 0.000, C 0.000 }
gfCNCPoint2[2069] = {X 308.3762, Y 86.2464, Z -2.1667, A 0.000, B 0.000, C 0.000 }
gfCNCPoint2[2070] = {X 308.3164, Y 84.6159, Z -2.1667, A 0.000, B 0.000, C 0.000 }
gfCNCPoint2[2071] = {X 308.3176, Y 83.2313, Z -2.1667, A 0.000, B 0.000, C 0.000 }
gfCNCPoint2[2072] = {X 308.3176, Y 62.9244, Z -2.1667, A 0.000, B 0.000, C 0.000 }
gfCNCPoint2[2073] = {X 307.4749, Y 62.7737, Z -2.1667, A 0.000, B 0.000, C 0.000 }
gfCNCPoint2[2074] = {X 306.6835, Y 62.4471, Z -2.1667, A 0.000, B 0.000, C 0.000 }
gfCNCPoint2[2075] = {X 305.9797, Y 61.9596, Z -2.1667, A 0.000, B 0.000, C 0.000 }
gfCNCPoint2[2076] = {X 305.3958, Y 61.3335, Z -2.1667, A 0.000, B 0.000, C 0.000 }
gfCNCPoint2[2077] = {X 304.9585, Y 60.5975, Z -2.1667, A 0.000, B 0.000, C 0.000 }
gfCNCPoint2[2078] = {X 304.6878, Y 59.7853, Z -2.1667, A 0.000, B 0.000, C 0.000 }
gfCNCPoint2[2079] = {X 304.5962, Y 58.9340, Z -2.1667, A 0.000, B 0.000, C 0.000 }
gfCNCPoint2[2080] = {X 304.5962, Y 58.0000, Z -2.1667, A 0.000, B 0.000, C 0.000 }
gfCNCPoint2[2081] = {X 304.6965, Y 57.1099, Z -2.1667, A 0.000, B 0.000, C 0.000 }
gfCNCPoint2[2082] = {X 304.9923, Y 56.2645, Z -2.1667, A 0.000, B 0.000, C 0.000 }
gfCNCPoint2[2083] = {X 305.4689, Y 55.5060, Z -2.1667, A 0.000, B 0.000, C 0.000 }
gfCNCPoint2[2084] = {X 306.1023, Y 54.8727, Z -2.1667, A 0.000, B 0.000, C 0.000 }
gfCNCPoint2[2085] = {X 306.8607, Y 54.3961, Z -2.1667, A 0.000, B 0.000, C 0.000 }
gfCNCPoint2[2086] = {X 307.7061, Y 54.1003, Z -2.1667, A 0.000, B 0.000, C 0.000 }
gfCNCPoint2[2087] = {X 308.5962, Y 54.0000, Z -2.1667, A 0.000, B 0.000, C 0.000 }
gfCNCPoint2[2088] = {X 324.3107, Y 54.0000, Z -2.1667, A 0.000, B 0.000, C 0.000 }
gfCNCPoint2[2089] = {X 325.2008, Y 54.1003, Z -2.1667, A 0.000, B 0.000, C 0.000 }
gfCNCPoint2[2090] = {X 326.0462, Y 54.3961, Z -2.1667, A 0.000, B 0.000, C 0.000 }
gfCNCPoint2[2091] = {X 326.8046, Y 54.8727, Z -2.1667, A 0.000, B 0.000, C 0.000 }
gfCNCPoint2[2092] = {X 327.4380, Y 55.5060, Z -2.1667, A 0.000, B 0.000, C 0.000 }
gfCNCPoint2[2093] = {X 327.9146, Y 56.2645, Z -2.1667, A 0.000, B 0.000, C 0.000 }
gfCNCPoint2[2094] = {X 328.2104, Y 57.1099, Z -2.1667, A 0.000, B 0.000, C 0.000 }
gfCNCPoint2[2095] = {X 328.3107, Y 58.0000, Z -2.1667, A 0.000, B 0.000, C 0.000 }
gfCNCPoint2[2096] = {X 328.3107, Y 58.9341, Z -2.1667, A 0.000, B 0.000, C 0.000 }
gfCNCPoint2[2097] = {X 328.2148, Y 59.7843, Z -2.1667, A 0.000, B 0.000, C 0.000 }
gfCNCPoint2[2098] = {X 327.9421, Y 60.5953, Z -2.1667, A 0.000, B 0.000, C 0.000 }
gfCNCPoint2[2099] = {X 327.5046, Y 61.3306, Z -2.1667, A 0.000, B 0.000, C 0.000 }
gfCNCPoint2[2100] = {X 326.9221, Y 61.9573, Z -2.1667, A 0.000, B 0.000, C 0.000 }
gfCNCPoint2[2101] = {X 326.2207, Y 62.4473, Z -2.1667, A 0.000, B 0.000, C 0.000 }
gfCNCPoint2[2102] = {X 325.4318, Y 62.7785, Z -2.1667, A 0.000, B 0.000, C 0.000 }
gfCNCPoint2[2103] = {X 324.5908, Y 62.9362, Z -2.1667, A 0.000, B 0.000, C 0.000 }
gfCNCPoint2[2104] = {X 324.5922, Y 83.2313, Z -2.1667, A 0.000, B 0.000, C 0.000 }
gfCNCPoint2[2105] = {X 324.6058, Y 84.6159, Z -2.1667, A 0.000, B 0.000, C 0.000 }
gfCNCPoint2[2106] = {X 324.6891, Y 85.9183, Z -2.1667, A 0.000, B 0.000, C 0.000 }
gfCNCPoint2[2107] = {X 324.9294, Y 87.2010, Z -2.1667, A 0.000, B 0.000, C 0.000 }
gfCNCPoint2[2108] = {X 325.2359, Y 87.5557, Z -2.1667, A 0.000, B 0.000, C 0.000 }
gfCNCPoint2[2109] = {X 325.6219, Y 87.8216, Z -2.1667, A 0.000, B 0.000, C 0.000 }
gfCNCPoint2[2110] = {X 326.0753, Y 88.0775, Z -2.1667, A 0.000, B 0.000, C 0.000 }
gfCNCPoint2[2111] = {X 327.5504, Y 88.6914, Z -2.1667, A 0.000, B 0.000, C 0.000 }
gfCNCPoint2[2112] = {X 329.0843, Y 89.1387, Z -2.1667, A 0.000, B 0.000, C 0.000 }
gfCNCPoint2[2113] = {X 332.1822, Y 89.7588, Z -2.1667, A 0.000, B 0.000, C 0.000 }
gfCNCPoint2[2114] = {X 335.3167, Y 90.1540, Z -2.1667, A 0.000, B 0.000, C 0.000 }
gfCNCPoint2[2115] = {X 339.4647, Y 90.4739, Z -2.1667, A 0.000, B 0.000, C 0.000 }
gfCNCPoint2[2116] = {X 343.6212, Y 90.6541, Z -2.1667, A 0.000, B 0.000, C 0.000 }
gfCNCPoint2[2117] = {X 347.7814, Y 90.6944, Z -2.1667, A 0.000, B 0.000, C 0.000 }
gfCNCPoint2[2118] = {X 352.1732, Y 90.6558, Z -2.1667, A 0.000, B 0.000, C 0.000 }
gfCNCPoint2[2119] = {X 356.5609, Y 90.4594, Z -2.1667, A 0.000, B 0.000, C 0.000 }
gfCNCPoint2[2120] = {X 360.9386, Y 90.1055, Z -2.1667, A 0.000, B 0.000, C 0.000 }
gfCNCPoint2[2121] = {X 363.2713, Y 89.8153, Z -2.1667, A 0.000, B 0.000, C 0.000 }
gfCNCPoint2[2122] = {X 365.5824, Y 89.3855, Z -2.1667, A 0.000, B 0.000, C 0.000 }
gfCNCPoint2[2123] = {X 367.8634, Y 88.8175, Z -2.1667, A 0.000, B 0.000, C 0.000 }
gfCNCPoint2[2124] = {X 368.8290, Y 88.4927, Z -2.1667, A 0.000, B 0.000, C 0.000 }
gfCNCPoint2[2125] = {X 369.7521, Y 88.0618, Z -2.1667, A 0.000, B 0.000, C 0.000 }
gfCNCPoint2[2126] = {X 370.6211, Y 87.5300, Z -2.1667, A 0.000, B 0.000, C 0.000 }
gfCNCPoint2[2127] = {X 370.8591, Y 87.2822, Z -2.1667, A 0.000, B 0.000, C 0.000 }
gfCNCPoint2[2128] = {X 370.9819, Y 86.9612, Z -2.1667, A 0.000, B 0.000, C 0.000 }
gfCNCPoint2[2129] = {X 371.1762, Y 85.3998, Z -2.1667, A 0.000, B 0.000, C 0.000 }
gfCNCPoint2[2130] = {X 371.2411, Y 83.8278, Z -2.1667, A 0.000, B 0.000, C 0.000 }
gfCNCPoint2[2131] = {X 371.2394, Y 63.0385, Z -2.1667, A 0.000, B 0.000, C 0.000 }
gfCNCPoint2[2132] = {X 371.2440, Y 62.9246, Z -2.1667, A 0.000, B 0.000, C 0.000 }
gfCNCPoint2[2133] = {X 371.0722, Y 62.9090, Z -2.1667, A 0.000, B 0.000, C 0.000 }
gfCNCPoint2[2134] = {X 370.9012, Y 62.8860, Z -2.1667, A 0.000, B 0.000, C 0.000 }
gfCNCPoint2[2135] = {X 369.9945, Y 62.6321, Z -2.1667, A 0.000, B 0.000, C 0.000 }
gfCNCPoint2[2136] = {X 369.1723, Y 62.1732, Z -2.1667, A 0.000, B 0.000, C 0.000 }
gfCNCPoint2[2137] = {X 368.4802, Y 61.5348, Z -2.1667, A 0.000, B 0.000, C 0.000 }
gfCNCPoint2[2138] = {X 367.9564, Y 60.7523, Z -2.1667, A 0.000, B 0.000, C 0.000 }
gfCNCPoint2[2139] = {X 367.6301, Y 59.8691, Z -2.1667, A 0.000, B 0.000, C 0.000 }
gfCNCPoint2[2140] = {X 367.5193, Y 58.9340, Z -2.1667, A 0.000, B 0.000, C 0.000 }
gfCNCPoint2[2141] = {X 367.5193, Y 58.0000, Z -2.1667, A 0.000, B 0.000, C 0.000 }
gfCNCPoint2[2142] = {X 367.6196, Y 57.1099, Z -2.1667, A 0.000, B 0.000, C 0.000 }
gfCNCPoint2[2143] = {X 367.9154, Y 56.2645, Z -2.1667, A 0.000, B 0.000, C 0.000 }
gfCNCPoint2[2144] = {X 368.3920, Y 55.5060, Z -2.1667, A 0.000, B 0.000, C 0.000 }
gfCNCPoint2[2145] = {X 369.0253, Y 54.8727, Z -2.1667, A 0.000, B 0.000, C 0.000 }
gfCNCPoint2[2146] = {X 369.7837, Y 54.3961, Z -2.1667, A 0.000, B 0.000, C 0.000 }
gfCNCPoint2[2147] = {X 370.6292, Y 54.1003, Z -2.1667, A 0.000, B 0.000, C 0.000 }
gfCNCPoint2[2148] = {X 371.5193, Y 54.0000, Z -2.1667, A 0.000, B 0.000, C 0.000 }
gfCNCPoint2[2149] = {X 388.0597, Y 54.0000, Z -2.1667, A 0.000, B 0.000, C 0.000 }
gfCNCPoint2[2150] = {X 388.9498, Y 54.1003, Z -2.1667, A 0.000, B 0.000, C 0.000 }
gfCNCPoint2[2151] = {X 389.7952, Y 54.3961, Z -2.1667, A 0.000, B 0.000, C 0.000 }
gfCNCPoint2[2152] = {X 390.5536, Y 54.8727, Z -2.1667, A 0.000, B 0.000, C 0.000 }
gfCNCPoint2[2153] = {X 391.1870, Y 55.5060, Z -2.1667, A 0.000, B 0.000, C 0.000 }
gfCNCPoint2[2154] = {X 391.6636, Y 56.2645, Z -2.1667, A 0.000, B 0.000, C 0.000 }
gfCNCPoint2[2155] = {X 391.9594, Y 57.1099, Z -2.1667, A 0.000, B 0.000, C 0.000 }
gfCNCPoint2[2156] = {X 392.0597, Y 58.0000, Z -2.1667, A 0.000, B 0.000, C 0.000 }
gfCNCPoint2[2157] = {X 392.0595, Y 58.9671, Z -2.1667, A 0.000, B 0.000, C 0.000 }
gfCNCPoint2[2158] = {X 391.9488, Y 59.8692, Z -2.1667, A 0.000, B 0.000, C 0.000 }
gfCNCPoint2[2159] = {X 391.6374, Y 60.7230, Z -2.1667, A 0.000, B 0.000, C 0.000 }
gfCNCPoint2[2160] = {X 391.1141, Y 61.5177, Z -2.1667, A 0.000, B 0.000, C 0.000 }
gfCNCPoint2[2161] = {X 390.4187, Y 62.1673, Z -2.1667, A 0.000, B 0.000, C 0.000 }
gfCNCPoint2[2162] = {X 389.5902, Y 62.6352, Z -2.1667, A 0.000, B 0.000, C 0.000 }
gfCNCPoint2[2163] = {X 388.6749, Y 62.8954, Z -2.1667, A 0.000, B 0.000, C 0.000 }
gfCNCPoint2[2164] = {X 388.5087, Y 62.9183, Z -2.1667, A 0.000, B 0.000, C 0.000 }
gfCNCPoint2[2165] = {X 388.3417, Y 62.9344, Z -2.1667, A 0.000, B 0.000, C 0.000 }
gfCNCPoint2[2166] = {X 388.3380, Y 63.1540, Z -2.1667, A 0.000, B 0.000, C 0.000 }
gfCNCPoint2[2167] = {X 388.3380, Y 83.9236, Z -2.1667, A 0.000, B 0.000, C 0.000 }
gfCNCPoint2[2168] = {X 388.3359, Y 84.6159, Z -2.1667, A 0.000, B 0.000, C 0.000 }
gfCNCPoint2[2169] = {X 388.2768, Y 86.2467, Z -2.1667, A 0.000, B 0.000, C 0.000 }
gfCNCPoint2[2170] = {X 388.0759, Y 87.8662, Z -2.1667, A 0.000, B 0.000, C 0.000 }
gfCNCPoint2[2171] = {X 387.7347, Y 89.4621, Z -2.1667, A 0.000, B 0.000, C 0.000 }
gfCNCPoint2[2172] = {X 387.2170, Y 91.0069, Z -2.1667, A 0.000, B 0.000, C 0.000 }
gfCNCPoint2[2173] = {X 386.4876, Y 92.4637, Z -2.1667, A 0.000, B 0.000, C 0.000 }
gfCNCPoint2[2174] = {X 385.5610, Y 93.8038, Z -2.1667, A 0.000, B 0.000, C 0.000 }
gfCNCPoint2[2175] = {X 384.4556, Y 95.0007, Z -2.1667, A 0.000, B 0.000, C 0.000 }
gfCNCPoint2[2176] = {X 382.9675, Y 96.2543, Z -2.1667, A 0.000, B 0.000, C 0.000 }
gfCNCPoint2[2177] = {X 381.3548, Y 97.3429, Z -2.1667, A 0.000, B 0.000, C 0.000 }
gfCNCPoint2[2178] = {X 379.6357, Y 98.2543, Z -2.1667, A 0.000, B 0.000, C 0.000 }
gfCNCPoint2[2179] = {X 377.3857, Y 99.2015, Z -2.1667, A 0.000, B 0.000, C 0.000 }
gfCNCPoint2[2180] = {X 375.0734, Y 99.9844, Z -2.1667, A 0.000, B 0.000, C 0.000 }
gfCNCPoint2[2181] = {X 372.7108, Y 100.5989, Z -2.1667, A 0.000, B 0.000, C 0.000 }
gfCNCPoint2[2182] = {X 368.9146, Y 101.3333, Z -2.1667, A 0.000, B 0.000, C 0.000 }
gfCNCPoint2[2183] = {X 365.0874, Y 101.8844, Z -2.1667, A 0.000, B 0.000, C 0.000 }
gfCNCPoint2[2184] = {X 361.2381, Y 102.2508, Z -2.1667, A 0.000, B 0.000, C 0.000 }
gfCNCPoint2[2185] = {X 357.2380, Y 102.4911, Z -2.1667, A 0.000, B 0.000, C 0.000 }
gfCNCPoint2[2186] = {X 353.2337, Y 102.6443, Z -2.1667, A 0.000, B 0.000, C 0.000 }
gfCNCPoint2[2187] = {X 353.3453, Y 106.7228, Z -2.1667, A 0.000, B 0.000, C 0.000 }
gfCNCPoint2[2188] = {X 353.3453, Y 106.7228, Z 0.8333, A 0.000, B 0.000, C 0.000 }
gfCNCPoint2[2189] = {X 353.3453, Y 106.7228, Z 11.0000, A 0.000, B 0.000, C 0.000 }
gfCNCPoint2[2190] = {X 411.5992, Y 79.5932, Z 11.0000, A 0.000, B 0.000, C 0.000 }
gfCNCPoint2[2191] = {X 411.5992, Y 79.5932, Z 0.8333, A 0.000, B 0.000, C 0.000 }
gfCNCPoint2[2192] = {X 411.5992, Y 79.5932, Z -2.1667, A 0.000, B 0.000, C 0.000 }
gfCNCPoint2[2193] = {X 413.7996, Y 83.0290, Z -2.1667, A 0.000, B 0.000, C 0.000 }
gfCNCPoint2[2194] = {X 428.0555, Y 73.8994, Z -2.1667, A 0.000, B 0.000, C 0.000 }
gfCNCPoint2[2195] = {X 403.7555, Y 64.3648, Z -2.1667, A 0.000, B 0.000, C 0.000 }
gfCNCPoint2[2196] = {X 402.0596, Y 63.8033, Z -2.1667, A 0.000, B 0.000, C 0.000 }
gfCNCPoint2[2197] = {X 400.3124, Y 63.4316, Z -2.1667, A 0.000, B 0.000, C 0.000 }
gfCNCPoint2[2198] = {X 398.5349, Y 63.2540, Z -2.1667, A 0.000, B 0.000, C 0.000 }
gfCNCPoint2[2199] = {X 397.5823, Y 63.1425, Z -2.1667, A 0.000, B 0.000, C 0.000 }
gfCNCPoint2[2200] = {X 396.6778, Y 62.8236, Z -2.1667, A 0.000, B 0.000, C 0.000 }
gfCNCPoint2[2201] = {X 395.8660, Y 62.3130, Z -2.1667, A 0.000, B 0.000, C 0.000 }
gfCNCPoint2[2202] = {X 395.1868, Y 61.6358, Z -2.1667, A 0.000, B 0.000, C 0.000 }
gfCNCPoint2[2203] = {X 394.6738, Y 60.8255, Z -2.1667, A 0.000, B 0.000, C 0.000 }
gfCNCPoint2[2204] = {X 394.3522, Y 59.9220, Z -2.1667, A 0.000, B 0.000, C 0.000 }
gfCNCPoint2[2205] = {X 394.2379, Y 58.9697, Z -2.1667, A 0.000, B 0.000, C 0.000 }
gfCNCPoint2[2206] = {X 394.2377, Y 58.0000, Z -2.1667, A 0.000, B 0.000, C 0.000 }
gfCNCPoint2[2207] = {X 394.3460, Y 57.0387, Z -2.1667, A 0.000, B 0.000, C 0.000 }
gfCNCPoint2[2208] = {X 394.6655, Y 56.1256, Z -2.1667, A 0.000, B 0.000, C 0.000 }
gfCNCPoint2[2209] = {X 395.1802, Y 55.3065, Z -2.1667, A 0.000, B 0.000, C 0.000 }
gfCNCPoint2[2210] = {X 395.8642, Y 54.6225, Z -2.1667, A 0.000, B 0.000, C 0.000 }
gfCNCPoint2[2211] = {X 396.6833, Y 54.1078, Z -2.1667, A 0.000, B 0.000, C 0.000 }
gfCNCPoint2[2212] = {X 397.5964, Y 53.7883, Z -2.1667, A 0.000, B 0.000, C 0.000 }
gfCNCPoint2[2213] = {X 398.5577, Y 53.6800, Z -2.1667, A 0.000, B 0.000, C 0.000 }
gfCNCPoint2[2214] = {X 419.4886, Y 53.6800, Z -2.1667, A 0.000, B 0.000, C 0.000 }
gfCNCPoint2[2215] = {X 420.4499, Y 53.7883, Z -2.1667, A 0.000, B 0.000, C 0.000 }
gfCNCPoint2[2216] = {X 421.3630, Y 54.1078, Z -2.1667, A 0.000, B 0.000, C 0.000 }
gfCNCPoint2[2217] = {X 422.1821, Y 54.6225, Z -2.1667, A 0.000, B 0.000, C 0.000 }
gfCNCPoint2[2218] = {X 422.8661, Y 55.3065, Z -2.1667, A 0.000, B 0.000, C 0.000 }
gfCNCPoint2[2219] = {X 423.3808, Y 56.1256, Z -2.1667, A 0.000, B 0.000, C 0.000 }
gfCNCPoint2[2220] = {X 423.7003, Y 57.0387, Z -2.1667, A 0.000, B 0.000, C 0.000 }
gfCNCPoint2[2221] = {X 423.8086, Y 58.0000, Z -2.1667, A 0.000, B 0.000, C 0.000 }
gfCNCPoint2[2222] = {X 423.8086, Y 58.2327, Z -2.1667, A 0.000, B 0.000, C 0.000 }
gfCNCPoint2[2223] = {X 429.6116, Y 60.4944, Z -2.1667, A 0.000, B 0.000, C 0.000 }
gfCNCPoint2[2224] = {X 457.8611, Y 71.7022, Z -2.1667, A 0.000, B 0.000, C 0.000 }
gfCNCPoint2[2225] = {X 457.8612, Y 63.2124, Z -2.1667, A 0.000, B 0.000, C 0.000 }
gfCNCPoint2[2226] = {X 457.0095, Y 63.0034, Z -2.1667, A 0.000, B 0.000, C 0.000 }
gfCNCPoint2[2227] = {X 456.2175, Y 62.6267, Z -2.1667, A 0.000, B 0.000, C 0.000 }
gfCNCPoint2[2228] = {X 455.5179, Y 62.0977, Z -2.1667, A 0.000, B 0.000, C 0.000 }
gfCNCPoint2[2229] = {X 454.9395, Y 61.4384, Z -2.1667, A 0.000, B 0.000, C 0.000 }
gfCNCPoint2[2230] = {X 454.5063, Y 60.6758, Z -2.1667, A 0.000, B 0.000, C 0.000 }
gfCNCPoint2[2231] = {X 454.2360, Y 59.8415, Z -2.1667, A 0.000, B 0.000, C 0.000 }
gfCNCPoint2[2232] = {X 454.1398, Y 58.9697, Z -2.1667, A 0.000, B 0.000, C 0.000 }
gfCNCPoint2[2233] = {X 454.1396, Y 58.0000, Z -2.1667, A 0.000, B 0.000, C 0.000 }
gfCNCPoint2[2234] = {X 454.2479, Y 57.0387, Z -2.1667, A 0.000, B 0.000, C 0.000 }
gfCNCPoint2[2235] = {X 454.5674, Y 56.1256, Z -2.1667, A 0.000, B 0.000, C 0.000 }
gfCNCPoint2[2236] = {X 455.0821, Y 55.3065, Z -2.1667, A 0.000, B 0.000, C 0.000 }
gfCNCPoint2[2237] = {X 455.7661, Y 54.6225, Z -2.1667, A 0.000, B 0.000, C 0.000 }
gfCNCPoint2[2238] = {X 456.5852, Y 54.1078, Z -2.1667, A 0.000, B 0.000, C 0.000 }
gfCNCPoint2[2239] = {X 457.4983, Y 53.7883, Z -2.1667, A 0.000, B 0.000, C 0.000 }
gfCNCPoint2[2240] = {X 458.4596, Y 53.6800, Z -2.1667, A 0.000, B 0.000, C 0.000 }
gfCNCPoint2[2241] = {X 475.0000, Y 53.6800, Z -2.1667, A 0.000, B 0.000, C 0.000 }
gfCNCPoint2[2242] = {X 475.9613, Y 53.7883, Z -2.1667, A 0.000, B 0.000, C 0.000 }
gfCNCPoint2[2243] = {X 476.8744, Y 54.1078, Z -2.1667, A 0.000, B 0.000, C 0.000 }
gfCNCPoint2[2244] = {X 477.6935, Y 54.6225, Z -2.1667, A 0.000, B 0.000, C 0.000 }
gfCNCPoint2[2245] = {X 478.3775, Y 55.3065, Z -2.1667, A 0.000, B 0.000, C 0.000 }
gfCNCPoint2[2246] = {X 478.8922, Y 56.1256, Z -2.1667, A 0.000, B 0.000, C 0.000 }
gfCNCPoint2[2247] = {X 479.2117, Y 57.0387, Z -2.1667, A 0.000, B 0.000, C 0.000 }
gfCNCPoint2[2248] = {X 479.3200, Y 58.0000, Z -2.1667, A 0.000, B 0.000, C 0.000 }
gfCNCPoint2[2249] = {X 479.3200, Y 58.9342, Z -2.1667, A 0.000, B 0.000, C 0.000 }
gfCNCPoint2[2250] = {X 479.2299, Y 59.8115, Z -2.1667, A 0.000, B 0.000, C 0.000 }
gfCNCPoint2[2251] = {X 478.9636, Y 60.6523, Z -2.1667, A 0.000, B 0.000, C 0.000 }
gfCNCPoint2[2252] = {X 478.5321, Y 61.4214, Z -2.1667, A 0.000, B 0.000, C 0.000 }
gfCNCPoint2[2253] = {X 477.9533, Y 62.0869, Z -2.1667, A 0.000, B 0.000, C 0.000 }
gfCNCPoint2[2254] = {X 477.2515, Y 62.6210, Z -2.1667, A 0.000, B 0.000, C 0.000 }
gfCNCPoint2[2255] = {X 476.4558, Y 63.0014, Z -2.1667, A 0.000, B 0.000, C 0.000 }
gfCNCPoint2[2256] = {X 475.5995, Y 63.2123, Z -2.1667, A 0.000, B 0.000, C 0.000 }
gfCNCPoint2[2257] = {X 475.5999, Y 92.7688, Z -2.1667, A 0.000, B 0.000, C 0.000 }
gfCNCPoint2[2258] = {X 475.9959, Y 92.8679, Z -2.1667, A 0.000, B 0.000, C 0.000 }
gfCNCPoint2[2259] = {X 476.3862, Y 92.9872, Z -2.1667, A 0.000, B 0.000, C 0.000 }
gfCNCPoint2[2260] = {X 477.1983, Y 93.3560, Z -2.1667, A 0.000, B 0.000, C 0.000 }
gfCNCPoint2[2261] = {X 477.9166, Y 93.8847, Z -2.1667, A 0.000, B 0.000, C 0.000 }
gfCNCPoint2[2262] = {X 478.5102, Y 94.5503, Z -2.1667, A 0.000, B 0.000, C 0.000 }
gfCNCPoint2[2263] = {X 478.9535, Y 95.3242, Z -2.1667, A 0.000, B 0.000, C 0.000 }
gfCNCPoint2[2264] = {X 479.2274, Y 96.1730, Z -2.1667, A 0.000, B 0.000, C 0.000 }
gfCNCPoint2[2265] = {X 479.3200, Y 97.0600, Z -2.1667, A 0.000, B 0.000, C 0.000 }
gfCNCPoint2[2266] = {X 479.3200, Y 98.0000, Z -2.1667, A 0.000, B 0.000, C 0.000 }
gfCNCPoint2[2267] = {X 479.2117, Y 98.9613, Z -2.1667, A 0.000, B 0.000, C 0.000 }
gfCNCPoint2[2268] = {X 478.8922, Y 99.8744, Z -2.1667, A 0.000, B 0.000, C 0.000 }
gfCNCPoint2[2269] = {X 478.3775, Y 100.6935, Z -2.1667, A 0.000, B 0.000, C 0.000 }
gfCNCPoint2[2270] = {X 477.6935, Y 101.3775, Z -2.1667, A 0.000, B 0.000, C 0.000 }
gfCNCPoint2[2271] = {X 476.8744, Y 101.8922, Z -2.1667, A 0.000, B 0.000, C 0.000 }
gfCNCPoint2[2272] = {X 475.9613, Y 102.2117, Z -2.1667, A 0.000, B 0.000, C 0.000 }
gfCNCPoint2[2273] = {X 475.0000, Y 102.3200, Z -2.1667, A 0.000, B 0.000, C 0.000 }
gfCNCPoint2[2274] = {X 458.4596, Y 102.3200, Z -2.1667, A 0.000, B 0.000, C 0.000 }
gfCNCPoint2[2275] = {X 457.4983, Y 102.2117, Z -2.1667, A 0.000, B 0.000, C 0.000 }
gfCNCPoint2[2276] = {X 456.5852, Y 101.8922, Z -2.1667, A 0.000, B 0.000, C 0.000 }
gfCNCPoint2[2277] = {X 455.7661, Y 101.3775, Z -2.1667, A 0.000, B 0.000, C 0.000 }
gfCNCPoint2[2278] = {X 455.0821, Y 100.6935, Z -2.1667, A 0.000, B 0.000, C 0.000 }
gfCNCPoint2[2279] = {X 454.5674, Y 99.8744, Z -2.1667, A 0.000, B 0.000, C 0.000 }
gfCNCPoint2[2280] = {X 454.2479, Y 98.9613, Z -2.1667, A 0.000, B 0.000, C 0.000 }
gfCNCPoint2[2281] = {X 454.1396, Y 98.0000, Z -2.1667, A 0.000, B 0.000, C 0.000 }
gfCNCPoint2[2282] = {X 454.1396, Y 97.0659, Z -2.1667, A 0.000, B 0.000, C 0.000 }
gfCNCPoint2[2283] = {X 454.2295, Y 96.1891, Z -2.1667, A 0.000, B 0.000, C 0.000 }
gfCNCPoint2[2284] = {X 454.4955, Y 95.3488, Z -2.1667, A 0.000, B 0.000, C 0.000 }
gfCNCPoint2[2285] = {X 454.9265, Y 94.5800, Z -2.1667, A 0.000, B 0.000, C 0.000 }
gfCNCPoint2[2286] = {X 455.5046, Y 93.9147, Z -2.1667, A 0.000, B 0.000, C 0.000 }
gfCNCPoint2[2287] = {X 456.2057, Y 93.3805, Z -2.1667, A 0.000, B 0.000, C 0.000 }
gfCNCPoint2[2288] = {X 457.0006, Y 92.9998, Z -2.1667, A 0.000, B 0.000, C 0.000 }
gfCNCPoint2[2289] = {X 457.8563, Y 92.7883, Z -2.1667, A 0.000, B 0.000, C 0.000 }
gfCNCPoint2[2290] = {X 457.8563, Y 85.5950, Z -2.1667, A 0.000, B 0.000, C 0.000 }
gfCNCPoint2[2291] = {X 444.8581, Y 80.4997, Z -2.1667, A 0.000, B 0.000, C 0.000 }
gfCNCPoint2[2292] = {X 420.0227, Y 96.5880, Z -2.1667, A 0.000, B 0.000, C 0.000 }
gfCNCPoint2[2293] = {X 420.0267, Y 97.0646, Z -2.1667, A 0.000, B 0.000, C 0.000 }
gfCNCPoint2[2294] = {X 420.0267, Y 98.0000, Z -2.1667, A 0.000, B 0.000, C 0.000 }
gfCNCPoint2[2295] = {X 419.9184, Y 98.9613, Z -2.1667, A 0.000, B 0.000, C 0.000 }
gfCNCPoint2[2296] = {X 419.5989, Y 99.8744, Z -2.1667, A 0.000, B 0.000, C 0.000 }
gfCNCPoint2[2297] = {X 419.0842, Y 100.6935, Z -2.1667, A 0.000, B 0.000, C 0.000 }
gfCNCPoint2[2298] = {X 418.4002, Y 101.3775, Z -2.1667, A 0.000, B 0.000, C 0.000 }
gfCNCPoint2[2299] = {X 417.5811, Y 101.8922, Z -2.1667, A 0.000, B 0.000, C 0.000 }
gfCNCPoint2[2300] = {X 416.6680, Y 102.2117, Z -2.1667, A 0.000, B 0.000, C 0.000 }
gfCNCPoint2[2301] = {X 415.7067, Y 102.3200, Z -2.1667, A 0.000, B 0.000, C 0.000 }
gfCNCPoint2[2302] = {X 396.4059, Y 102.3200, Z -2.1667, A 0.000, B 0.000, C 0.000 }
gfCNCPoint2[2303] = {X 395.4447, Y 102.2117, Z -2.1667, A 0.000, B 0.000, C 0.000 }
gfCNCPoint2[2304] = {X 394.5316, Y 101.8922, Z -2.1667, A 0.000, B 0.000, C 0.000 }
gfCNCPoint2[2305] = {X 393.7125, Y 101.3775, Z -2.1667, A 0.000, B 0.000, C 0.000 }
gfCNCPoint2[2306] = {X 393.0284, Y 100.6935, Z -2.1667, A 0.000, B 0.000, C 0.000 }
gfCNCPoint2[2307] = {X 392.5138, Y 99.8744, Z -2.1667, A 0.000, B 0.000, C 0.000 }
gfCNCPoint2[2308] = {X 392.1943, Y 98.9613, Z -2.1667, A 0.000, B 0.000, C 0.000 }
gfCNCPoint2[2309] = {X 392.0859, Y 98.0000, Z -2.1667, A 0.000, B 0.000, C 0.000 }
gfCNCPoint2[2310] = {X 392.0859, Y 97.0659, Z -2.1667, A 0.000, B 0.000, C 0.000 }
gfCNCPoint2[2311] = {X 392.1938, Y 96.1069, Z -2.1667, A 0.000, B 0.000, C 0.000 }
gfCNCPoint2[2312] = {X 392.5118, Y 95.1956, Z -2.1667, A 0.000, B 0.000, C 0.000 }
gfCNCPoint2[2313] = {X 393.0242, Y 94.3778, Z -2.1667, A 0.000, B 0.000, C 0.000 }
gfCNCPoint2[2314] = {X 393.7054, Y 93.6941, Z -2.1667, A 0.000, B 0.000, C 0.000 }
gfCNCPoint2[2315] = {X 394.5214, Y 93.1787, Z -2.1667, A 0.000, B 0.000, C 0.000 }
gfCNCPoint2[2316] = {X 395.4314, Y 92.8573, Z -2.1667, A 0.000, B 0.000, C 0.000 }
gfCNCPoint2[2317] = {X 396.3901, Y 92.7460, Z -2.1667, A 0.000, B 0.000, C 0.000 }
gfCNCPoint2[2318] = {X 397.3434, Y 92.7056, Z -2.1667, A 0.000, B 0.000, C 0.000 }
gfCNCPoint2[2319] = {X 398.2933, Y 92.6153, Z -2.1667, A 0.000, B 0.000, C 0.000 }
gfCNCPoint2[2320] = {X 398.9443, Y 92.4577, Z -2.1667, A 0.000, B 0.000, C 0.000 }
gfCNCPoint2[2321] = {X 399.5436, Y 92.1587, Z -2.1667, A 0.000, B 0.000, C 0.000 }
gfCNCPoint2[2322] = {X 413.7996, Y 83.0290, Z -2.1667, A 0.000, B 0.000, C 0.000 }
gfCNCPoint2[2323] = {X 411.6424, Y 79.6606, Z -2.1667, A 0.000, B 0.000, C 0.000 }
gfCNCPoint2[2324] = {X 413.8427, Y 83.0964, Z -2.1667, A 0.000, B 0.000, C 0.000 }
gfCNCPoint2[2325] = {X 428.2307, Y 73.8822, Z -2.1667, A 0.000, B 0.000, C 0.000 }
gfCNCPoint2[2326] = {X 403.7847, Y 64.2904, Z -2.1667, A 0.000, B 0.000, C 0.000 }
gfCNCPoint2[2327] = {X 402.0801, Y 63.7260, Z -2.1667, A 0.000, B 0.000, C 0.000 }
gfCNCPoint2[2328] = {X 400.3237, Y 63.3524, Z -2.1667, A 0.000, B 0.000, C 0.000 }
gfCNCPoint2[2329] = {X 398.5369, Y 63.1740, Z -2.1667, A 0.000, B 0.000, C 0.000 }
gfCNCPoint2[2330] = {X 397.6017, Y 63.0649, Z -2.1667, A 0.000, B 0.000, C 0.000 }
gfCNCPoint2[2331] = {X 396.7136, Y 62.7520, Z -2.1667, A 0.000, B 0.000, C 0.000 }
gfCNCPoint2[2332] = {X 395.9165, Y 62.2510, Z -2.1667, A 0.000, B 0.000, C 0.000 }
gfCNCPoint2[2333] = {X 395.2497, Y 61.5863, Z -2.1667, A 0.000, B 0.000, C 0.000 }
gfCNCPoint2[2334] = {X 394.7459, Y 60.7909, Z -2.1667, A 0.000, B 0.000, C 0.000 }
gfCNCPoint2[2335] = {X 394.4301, Y 59.9039, Z -2.1667, A 0.000, B 0.000, C 0.000 }
gfCNCPoint2[2336] = {X 394.3179, Y 58.9691, Z -2.1667, A 0.000, B 0.000, C 0.000 }
gfCNCPoint2[2337] = {X 394.3177, Y 58.0000, Z -2.1667, A 0.000, B 0.000, C 0.000 }
gfCNCPoint2[2338] = {X 394.4240, Y 57.0565, Z -2.1667, A 0.000, B 0.000, C 0.000 }
gfCNCPoint2[2339] = {X 394.7376, Y 56.1603, Z -2.1667, A 0.000, B 0.000, C 0.000 }
gfCNCPoint2[2340] = {X 395.2428, Y 55.3564, Z -2.1667, A 0.000, B 0.000, C 0.000 }
gfCNCPoint2[2341] = {X 395.9141, Y 54.6850, Z -2.1667, A 0.000, B 0.000, C 0.000 }
gfCNCPoint2[2342] = {X 396.7181, Y 54.1799, Z -2.1667, A 0.000, B 0.000, C 0.000 }
gfCNCPoint2[2343] = {X 397.6142, Y 53.8663, Z -2.1667, A 0.000, B 0.000, C 0.000 }
gfCNCPoint2[2344] = {X 398.5577, Y 53.7600, Z -2.1667, A 0.000, B 0.000, C 0.000 }
gfCNCPoint2[2345] = {X 419.4886, Y 53.7600, Z -2.1667, A 0.000, B 0.000, C 0.000 }
gfCNCPoint2[2346] = {X 420.4321, Y 53.8663, Z -2.1667, A 0.000, B 0.000, C 0.000 }
gfCNCPoint2[2347] = {X 421.3283, Y 54.1799, Z -2.1667, A 0.000, B 0.000, C 0.000 }
gfCNCPoint2[2348] = {X 422.1322, Y 54.6850, Z -2.1667, A 0.000, B 0.000, C 0.000 }
gfCNCPoint2[2349] = {X 422.8036, Y 55.3564, Z -2.1667, A 0.000, B 0.000, C 0.000 }
gfCNCPoint2[2350] = {X 423.3087, Y 56.1603, Z -2.1667, A 0.000, B 0.000, C 0.000 }
gfCNCPoint2[2351] = {X 423.6223, Y 57.0565, Z -2.1667, A 0.000, B 0.000, C 0.000 }
gfCNCPoint2[2352] = {X 423.7286, Y 58.0000, Z -2.1667, A 0.000, B 0.000, C 0.000 }
gfCNCPoint2[2353] = {X 423.7286, Y 58.2874, Z -2.1667, A 0.000, B 0.000, C 0.000 }
gfCNCPoint2[2354] = {X 429.5823, Y 60.5688, Z -2.1667, A 0.000, B 0.000, C 0.000 }
gfCNCPoint2[2355] = {X 457.9411, Y 71.8200, Z -2.1667, A 0.000, B 0.000, C 0.000 }
gfCNCPoint2[2356] = {X 457.9412, Y 63.1423, Z -2.1667, A 0.000, B 0.000, C 0.000 }
gfCNCPoint2[2357] = {X 457.0926, Y 62.9477, Z -2.1667, A 0.000, B 0.000, C 0.000 }
gfCNCPoint2[2358] = {X 456.3016, Y 62.5838, Z -2.1667, A 0.000, B 0.000, C 0.000 }
gfCNCPoint2[2359] = {X 455.6016, Y 62.0660, Z -2.1667, A 0.000, B 0.000, C 0.000 }
gfCNCPoint2[2360] = {X 455.0221, Y 61.4162, Z -2.1667, A 0.000, B 0.000, C 0.000 }
gfCNCPoint2[2361] = {X 454.5876, Y 60.6617, Z -2.1667, A 0.000, B 0.000, C 0.000 }
gfCNCPoint2[2362] = {X 454.3163, Y 59.8344, Z -2.1667, A 0.000, B 0.000, C 0.000 }
gfCNCPoint2[2363] = {X 454.2197, Y 58.9691, Z -2.1667, A 0.000, B 0.000, C 0.000 }
gfCNCPoint2[2364] = {X 454.2196, Y 58.0000, Z -2.1667, A 0.000, B 0.000, C 0.000 }
gfCNCPoint2[2365] = {X 454.3259, Y 57.0565, Z -2.1667, A 0.000, B 0.000, C 0.000 }
gfCNCPoint2[2366] = {X 454.6395, Y 56.1603, Z -2.1667, A 0.000, B 0.000, C 0.000 }
gfCNCPoint2[2367] = {X 455.1446, Y 55.3564, Z -2.1667, A 0.000, B 0.000, C 0.000 }
gfCNCPoint2[2368] = {X 455.8160, Y 54.6850, Z -2.1667, A 0.000, B 0.000, C 0.000 }
gfCNCPoint2[2369] = {X 456.6199, Y 54.1799, Z -2.1667, A 0.000, B 0.000, C 0.000 }
gfCNCPoint2[2370] = {X 457.5161, Y 53.8663, Z -2.1667, A 0.000, B 0.000, C 0.000 }
gfCNCPoint2[2371] = {X 458.4596, Y 53.7600, Z -2.1667, A 0.000, B 0.000, C 0.000 }
gfCNCPoint2[2372] = {X 475.0000, Y 53.7600, Z -2.1667, A 0.000, B 0.000, C 0.000 }
gfCNCPoint2[2373] = {X 475.9435, Y 53.8663, Z -2.1667, A 0.000, B 0.000, C 0.000 }
gfCNCPoint2[2374] = {X 476.8397, Y 54.1799, Z -2.1667, A 0.000, B 0.000, C 0.000 }
gfCNCPoint2[2375] = {X 477.6436, Y 54.6850, Z -2.1667, A 0.000, B 0.000, C 0.000 }
gfCNCPoint2[2376] = {X 478.3150, Y 55.3564, Z -2.1667, A 0.000, B 0.000, C 0.000 }
gfCNCPoint2[2377] = {X 478.8201, Y 56.1603, Z -2.1667, A 0.000, B 0.000, C 0.000 }
gfCNCPoint2[2378] = {X 479.1337, Y 57.0565, Z -2.1667, A 0.000, B 0.000, C 0.000 }
gfCNCPoint2[2379] = {X 479.2400, Y 58.0000, Z -2.1667, A 0.000, B 0.000, C 0.000 }
gfCNCPoint2[2380] = {X 479.2400, Y 58.9342, Z -2.1667, A 0.000, B 0.000, C 0.000 }
gfCNCPoint2[2381] = {X 479.1496, Y 59.8050, Z -2.1667, A 0.000, B 0.000, C 0.000 }
gfCNCPoint2[2382] = {X 478.8823, Y 60.6387, Z -2.1667, A 0.000, B 0.000, C 0.000 }
gfCNCPoint2[2383] = {X 478.4494, Y 61.3997, Z -2.1667, A 0.000, B 0.000, C 0.000 }
gfCNCPoint2[2384] = {X 477.8695, Y 62.0555, Z -2.1667, A 0.000, B 0.000, C 0.000 }
gfCNCPoint2[2385] = {X 477.1673, Y 62.5783, Z -2.1667, A 0.000, B 0.000, C 0.000 }
gfCNCPoint2[2386] = {X 476.3726, Y 62.9457, Z -2.1667, A 0.000, B 0.000, C 0.000 }
gfCNCPoint2[2387] = {X 475.5195, Y 63.1421, Z -2.1667, A 0.000, B 0.000, C 0.000 }
gfCNCPoint2[2388] = {X 475.5199, Y 92.8332, Z -2.1667, A 0.000, B 0.000, C 0.000 }
gfCNCPoint2[2389] = {X 475.9436, Y 92.9365, Z -2.1667, A 0.000, B 0.000, C 0.000 }
gfCNCPoint2[2390] = {X 476.3609, Y 93.0631, Z -2.1667, A 0.000, B 0.000, C 0.000 }
gfCNCPoint2[2391] = {X 477.1578, Y 93.4250, Z -2.1667, A 0.000, B 0.000, C 0.000 }
gfCNCPoint2[2392] = {X 477.8627, Y 93.9438, Z -2.1667, A 0.000, B 0.000, C 0.000 }
gfCNCPoint2[2393] = {X 478.4453, Y 94.5971, Z -2.1667, A 0.000, B 0.000, C 0.000 }
gfCNCPoint2[2394] = {X 478.8803, Y 95.3565, Z -2.1667, A 0.000, B 0.000, C 0.000 }
gfCNCPoint2[2395] = {X 479.1491, Y 96.1895, Z -2.1667, A 0.000, B 0.000, C 0.000 }
gfCNCPoint2[2396] = {X 479.2400, Y 97.0600, Z -2.1667, A 0.000, B 0.000, C 0.000 }
gfCNCPoint2[2397] = {X 479.2400, Y 98.0000, Z -2.1667, A 0.000, B 0.000, C 0.000 }
gfCNCPoint2[2398] = {X 479.1337, Y 98.9435, Z -2.1667, A 0.000, B 0.000, C 0.000 }
gfCNCPoint2[2399] = {X 478.8201, Y 99.8397, Z -2.1667, A 0.000, B 0.000, C 0.000 }
gfCNCPoint2[2400] = {X 478.3150, Y 100.6436, Z -2.1667, A 0.000, B 0.000, C 0.000 }
gfCNCPoint2[2401] = {X 477.6436, Y 101.3150, Z -2.1667, A 0.000, B 0.000, C 0.000 }
gfCNCPoint2[2402] = {X 476.8397, Y 101.8201, Z -2.1667, A 0.000, B 0.000, C 0.000 }
gfCNCPoint2[2403] = {X 475.9435, Y 102.1337, Z -2.1667, A 0.000, B 0.000, C 0.000 }
gfCNCPoint2[2404] = {X 475.0000, Y 102.2400, Z -2.1667, A 0.000, B 0.000, C 0.000 }
gfCNCPoint2[2405] = {X 458.4596, Y 102.2400, Z -2.1667, A 0.000, B 0.000, C 0.000 }
gfCNCPoint2[2406] = {X 457.5161, Y 102.1337, Z -2.1667, A 0.000, B 0.000, C 0.000 }
gfCNCPoint2[2407] = {X 456.6199, Y 101.8201, Z -2.1667, A 0.000, B 0.000, C 0.000 }
gfCNCPoint2[2408] = {X 455.8160, Y 101.3150, Z -2.1667, A 0.000, B 0.000, C 0.000 }
gfCNCPoint2[2409] = {X 455.1446, Y 100.6436, Z -2.1667, A 0.000, B 0.000, C 0.000 }
gfCNCPoint2[2410] = {X 454.6395, Y 99.8397, Z -2.1667, A 0.000, B 0.000, C 0.000 }
gfCNCPoint2[2411] = {X 454.3259, Y 98.9435, Z -2.1667, A 0.000, B 0.000, C 0.000 }
gfCNCPoint2[2412] = {X 454.2196, Y 98.0000, Z -2.1667, A 0.000, B 0.000, C 0.000 }
gfCNCPoint2[2413] = {X 454.2196, Y 97.0659, Z -2.1667, A 0.000, B 0.000, C 0.000 }
gfCNCPoint2[2414] = {X 454.3099, Y 96.1957, Z -2.1667, A 0.000, B 0.000, C 0.000 }
gfCNCPoint2[2415] = {X 454.5769, Y 95.3624, Z -2.1667, A 0.000, B 0.000, C 0.000 }
gfCNCPoint2[2416] = {X 455.0092, Y 94.6018, Z -2.1667, A 0.000, B 0.000, C 0.000 }
gfCNCPoint2[2417] = {X 455.5884, Y 93.9460, Z -2.1667, A 0.000, B 0.000, C 0.000 }
gfCNCPoint2[2418] = {X 456.2899, Y 93.4231, Z -2.1667, A 0.000, B 0.000, C 0.000 }
gfCNCPoint2[2419] = {X 457.0838, Y 93.0553, Z -2.1667, A 0.000, B 0.000, C 0.000 }
gfCNCPoint2[2420] = {X 457.9363, Y 92.8584, Z -2.1667, A 0.000, B 0.000, C 0.000 }
gfCNCPoint2[2421] = {X 457.9363, Y 85.5404, Z -2.1667, A 0.000, B 0.000, C 0.000 }
gfCNCPoint2[2422] = {X 444.8491, Y 80.4102, Z -2.1667, A 0.000, B 0.000, C 0.000 }
